LIN {X 0,Y 566.661,Z 389.019,A -85,B 0,C 180,E1 -2630.32,E2 -2630.32} C_VEL
LIN {X 0,Y 566.806,Z 374.387,A -85,B 0,C 180,E1 -2632.99,E2 -2632.99} C_VEL
LIN {X 0,Y 566.858,Z 367.103,A -85,B 0,C 180,E1 -2634.345,E2 -2634.345} C_VEL
LIN {X 0,Y 566.237,Z 363.511,A -85,B 0,C 180,E1 -2635.093,E2 -2635.093} C_VEL
LIN {X 0,Y 566.232,Z 363.455,A -85,B 0,C 180,E1 -2638.141,E2 -2638.141} C_VEL
LIN {X 0,Y 566.19,Z 363.456,A -85,B 0,C 180,E1 -2640.592,E2 -2640.592} C_VEL
LIN {X 0,Y 566.231,Z 363.447,A -85,B 0,C 180,E1 -2643.101,E2 -2643.101} C_VEL
LIN {X 0,Y 566.215,Z 363.454,A -85,B 0,C 180,E1 -2645.688,E2 -2645.688} C_VEL
LIN {X 0,Y 566.218,Z 363.451,A -85,B 0,C 180,E1 -2648.558,E2 -2648.558} C_VEL
LIN {X 0,Y 566.213,Z 363.446,A -85,B 0,C 180,E1 -2651.136,E2 -2651.136} C_VEL
LIN {X 0,Y 566.198,Z 363.46,A -85,B 0,C 180,E1 -2654.035,E2 -2654.035} C_VEL
LIN {X 0,Y 566.206,Z 363.45,A -85,B 0,C 180,E1 -2657.082,E2 -2657.082} C_VEL
LIN {X 0,Y 566.228,Z 363.455,A -85,B 0,C 180,E1 -2659.802,E2 -2659.802} C_VEL
LIN {X 0,Y 566.199,Z 363.452,A -85,B 0,C 180,E1 -2662.599,E2 -2662.599} C_VEL
LIN {X 0,Y 566.209,Z 363.449,A -85,B 0,C 180,E1 -2665.182,E2 -2665.182} C_VEL
LIN {X 0,Y 566.235,Z 363.453,A -85,B 0,C 180,E1 -2667.743,E2 -2667.743} C_VEL
LIN {X 0,Y 566.228,Z 363.45,A -85,B 0,C 180,E1 -2670.323,E2 -2670.323} C_VEL
LIN {X 0,Y 566.218,Z 363.446,A -85,B 0,C 180,E1 -2672.661,E2 -2672.661} C_VEL
LIN {X 0,Y 566.235,Z 363.445,A -85,B 0,C 180,E1 -2675.039,E2 -2675.039} C_VEL
LIN {X 0,Y 566.194,Z 363.455,A -85,B 0,C 180,E1 -2678.137,E2 -2678.137} C_VEL
LIN {X 0,Y 566.235,Z 363.443,A -85,B 0,C 180,E1 -2680.611,E2 -2680.611} C_VEL
LIN {X 0,Y 566.219,Z 363.45,A -85,B 0,C 180,E1 -2683.412,E2 -2683.412} C_VEL
LIN {X 0,Y 566.197,Z 363.452,A -85,B 0,C 180,E1 -2686.358,E2 -2686.358} C_VEL
LIN {X 0,Y 566.232,Z 363.445,A -85,B 0,C 180,E1 -2688.675,E2 -2688.675} C_VEL
LIN {X 0,Y 566.232,Z 363.446,A -85,B 0,C 180,E1 -2691.434,E2 -2691.434} C_VEL
LIN {X 0,Y 566.258,Z 363.445,A -85,B 0,C 180,E1 -2694.301,E2 -2694.301} C_VEL
LIN {X 0,Y 566.278,Z 363.445,A -85,B 0,C 180,E1 -2697.866,E2 -2697.866} C_VEL
LIN {X 0,Y 566.302,Z 363.433,A -85,B 0,C 180,E1 -2700.711,E2 -2700.711} C_VEL
LIN {X 0,Y 566.273,Z 363.441,A -85,B 0,C 180,E1 -2702.845,E2 -2702.845} C_VEL
LIN {X 0,Y 566.256,Z 363.452,A -85,B 0,C 180,E1 -2705.698,E2 -2705.698} C_VEL
LIN {X 0,Y 566.23,Z 363.444,A -85,B 0,C 180,E1 -2708.565,E2 -2708.565} C_VEL
LIN {X 0,Y 566.238,Z 363.45,A -85,B 0,C 180,E1 -2711.454,E2 -2711.454} C_VEL
LIN {X 0,Y 566.231,Z 363.447,A -85,B 0,C 180,E1 -2714.506,E2 -2714.506} C_VEL
LIN {X 0,Y 566.197,Z 363.457,A -85,B 0,C 180,E1 -2717.331,E2 -2717.331} C_VEL
LIN {X 0,Y 566.211,Z 363.447,A -85,B 0,C 180,E1 -2720.337,E2 -2720.337} C_VEL
LIN {X 0,Y 566.185,Z 363.462,A -85,B 0,C 180,E1 -2723.404,E2 -2723.404} C_VEL
LIN {X 0,Y 566.221,Z 363.451,A -85,B 0,C 180,E1 -2725.748,E2 -2725.748} C_VEL
LIN {X 0,Y 566.213,Z 363.453,A -85,B 0,C 180,E1 -2727.49,E2 -2727.49} C_VEL
LIN {X 0,Y 565.533,Z 363.534,A -85,B 0,C 180,E1 -2728.084,E2 -2728.084} C_VEL
LIN {X 0,Y 562.662,Z 363.893,A -85,B 0,C 180,E1 -2729.047,E2 -2729.047} C_VEL
LIN {X 0,Y 560.248,Z 364.196,A -85,B 0,C 180,E1 -2729.823,E2 -2729.823} C_VEL
LIN {X 0,Y 559.221,Z 364.321,A -85,B 0,C 180,E1 -2730.421,E2 -2730.421} C_VEL
LIN {X 0,Y 559.142,Z 364.331,A -85,B 0,C 180,E1 -2730.624,E2 -2730.624} C_VEL
LIN {X 0,Y 559.161,Z 364.332,A -85,B 0,C 180,E1 -2733.574,E2 -2733.574} C_VEL
LIN {X 0,Y 559.165,Z 364.327,A -85,B 0,C 180,E1 -2736.448,E2 -2736.448} C_VEL
LIN {X 0,Y 559.174,Z 364.33,A -85,B 0,C 180,E1 -2738.934,E2 -2738.934} C_VEL
LIN {X 0,Y 559.188,Z 364.328,A -85,B 0,C 180,E1 -2741.767,E2 -2741.767} C_VEL
LIN {X 0,Y 559.136,Z 364.333,A -85,B 0,C 180,E1 -2744.739,E2 -2744.739} C_VEL
LIN {X 0,Y 559.169,Z 364.321,A -85,B 0,C 180,E1 -2747.863,E2 -2747.863} C_VEL
LIN {X 0,Y 559.182,Z 364.324,A -85,B 0,C 180,E1 -2750.135,E2 -2750.135} C_VEL
LIN {X 0,Y 559.144,Z 364.335,A -85,B 0,C 180,E1 -2752.892,E2 -2752.892} C_VEL
LIN {X 0,Y 559.154,Z 364.331,A -85,B 0,C 180,E1 -2755.556,E2 -2755.556} C_VEL
LIN {X 0,Y 559.168,Z 364.328,A -85,B 0,C 180,E1 -2758.138,E2 -2758.138} C_VEL
LIN {X 0,Y 559.155,Z 364.328,A -85,B 0,C 180,E1 -2760.647,E2 -2760.647} C_VEL
LIN {X 0,Y 559.168,Z 364.337,A -85,B 0,C 180,E1 -2763.172,E2 -2763.172} C_VEL
LIN {X 0,Y 559.154,Z 364.335,A -85,B 0,C 180,E1 -2765.495,E2 -2765.495} C_VEL
LIN {X 0,Y 559.168,Z 364.33,A -85,B 0,C 180,E1 -2768.624,E2 -2768.624} C_VEL
LIN {X 0,Y 559.168,Z 364.335,A -85,B 0,C 180,E1 -2770.926,E2 -2770.926} C_VEL
LIN {X 0,Y 559.164,Z 364.329,A -85,B 0,C 180,E1 -2773.948,E2 -2773.948} C_VEL
LIN {X 0,Y 559.17,Z 364.328,A -85,B 0,C 180,E1 -2776.184,E2 -2776.184} C_VEL
LIN {X 0,Y 559.193,Z 364.334,A -85,B 0,C 180,E1 -2779.133,E2 -2779.133} C_VEL
LIN {X 0,Y 559.201,Z 364.324,A -85,B 0,C 180,E1 -2782.053,E2 -2782.053} C_VEL
LIN {X 0,Y 559.252,Z 364.326,A -85,B 0,C 180,E1 -2784.953,E2 -2784.953} C_VEL
LIN {X 0,Y 559.253,Z 364.318,A -85,B 0,C 180,E1 -2787.839,E2 -2787.839} C_VEL
LIN {X 0,Y 559.27,Z 364.321,A -85,B 0,C 180,E1 -2790.72,E2 -2790.72} C_VEL
LIN {X 0,Y 559.235,Z 364.328,A -85,B 0,C 180,E1 -2792.881,E2 -2792.881} C_VEL
LIN {X 0,Y 559.235,Z 364.32,A -85,B 0,C 180,E1 -2795.77,E2 -2795.77} C_VEL
LIN {X 0,Y 559.188,Z 364.332,A -85,B 0,C 180,E1 -2798.674,E2 -2798.674} C_VEL
LIN {X 0,Y 559.202,Z 364.325,A -85,B 0,C 180,E1 -2801.6,E2 -2801.6} C_VEL
LIN {X 0,Y 559.196,Z 364.33,A -85,B 0,C 180,E1 -2804.595,E2 -2804.595} C_VEL
LIN {X 0,Y 559.159,Z 364.33,A -85,B 0,C 180,E1 -2807.556,E2 -2807.556} C_VEL
LIN {X 0,Y 559.168,Z 364.328,A -85,B 0,C 180,E1 -2809.837,E2 -2809.837} C_VEL
LIN {X 0,Y 559.137,Z 364.333,A -85,B 0,C 180,E1 -2812.152,E2 -2812.152} C_VEL
LIN {X 0,Y 559.175,Z 364.331,A -85,B 0,C 180,E1 -2815.187,E2 -2815.187} C_VEL
LIN {X 0,Y 559.19,Z 364.325,A -85,B 0,C 180,E1 -2817.711,E2 -2817.711} C_VEL
LIN {X 0,Y 559.164,Z 364.327,A -85,B 0,C 180,E1 -2820.181,E2 -2820.181} C_VEL
LIN {X 0,Y 559.17,Z 364.336,A -85,B 0,C 180,E1 -2822.714,E2 -2822.714} C_VEL
LIN {X 0,Y 559.154,Z 364.328,A -85,B 0,C 180,E1 -2825.321,E2 -2825.321} C_VEL
LIN {X 0,Y 559.13,Z 364.333,A -85,B 0,C 180,E1 -2828.017,E2 -2828.017} C_VEL
LIN {X 0,Y 559.169,Z 364.328,A -85,B 0,C 180,E1 -2830.81,E2 -2830.81} C_VEL
LIN {X 0,Y 559.137,Z 364.327,A -85,B 0,C 180,E1 -2833.733,E2 -2833.733} C_VEL
LIN {X 0,Y 559.165,Z 364.335,A -85,B 0,C 180,E1 -2836.8,E2 -2836.8} C_VEL
LIN {X 0,Y 559.17,Z 364.327,A -85,B 0,C 180,E1 -2839.189,E2 -2839.189} C_VEL
LIN {X 0,Y 559.128,Z 364.334,A -85,B 0,C 180,E1 -2841.983,E2 -2841.983} C_VEL
LIN {X 0,Y 559.152,Z 364.333,A -85,B 0,C 180,E1 -2844.783,E2 -2844.783} C_VEL
LIN {X 0,Y 559.168,Z 364.327,A -85,B 0,C 180,E1 -2847.361,E2 -2847.361} C_VEL
LIN {X 0,Y 559.182,Z 364.329,A -85,B 0,C 180,E1 -2850.135,E2 -2850.135} C_VEL
LIN {X 0,Y 559.175,Z 364.325,A -85,B 0,C 180,E1 -2853.17,E2 -2853.17} C_VEL
LIN {X 0,Y 559.15,Z 364.329,A -85,B 0,C 180,E1 -2855.495,E2 -2855.495} C_VEL
LIN {X 0,Y 559.171,Z 364.332,A -85,B 0,C 180,E1 -2858.624,E2 -2858.624} C_VEL
LIN {X 0,Y 559.165,Z 364.326,A -85,B 0,C 180,E1 -2860.927,E2 -2860.927} C_VEL
LIN {X 0,Y 559.166,Z 364.329,A -85,B 0,C 180,E1 -2863.948,E2 -2863.948} C_VEL
LIN {X 0,Y 559.167,Z 364.333,A -85,B 0,C 180,E1 -2866.184,E2 -2866.184} C_VEL
LIN {X 0,Y 559.189,Z 364.32,A -85,B 0,C 180,E1 -2869.134,E2 -2869.134} C_VEL
LIN {X 0,Y 559.201,Z 364.324,A -85,B 0,C 180,E1 -2872.054,E2 -2872.054} C_VEL
LIN {X 0,Y 559.252,Z 364.318,A -85,B 0,C 180,E1 -2874.954,E2 -2874.954} C_VEL
LIN {X 0,Y 559.248,Z 364.317,A -85,B 0,C 180,E1 -2877.84,E2 -2877.84} C_VEL
LIN {X 0,Y 559.27,Z 364.316,A -85,B 0,C 180,E1 -2880.72,E2 -2880.72} C_VEL
LIN {X 0,Y 559.238,Z 364.32,A -85,B 0,C 180,E1 -2882.882,E2 -2882.882} C_VEL
LIN {X 0,Y 559.225,Z 364.322,A -85,B 0,C 180,E1 -2885.771,E2 -2885.771} C_VEL
LIN {X 0,Y 559.187,Z 364.322,A -85,B 0,C 180,E1 -2888.675,E2 -2888.675} C_VEL
LIN {X 0,Y 559.2,Z 364.321,A -85,B 0,C 180,E1 -2891.601,E2 -2891.601} C_VEL
LIN {X 0,Y 559.194,Z 364.327,A -85,B 0,C 180,E1 -2894.596,E2 -2894.596} C_VEL
LIN {X 0,Y 559.159,Z 364.326,A -85,B 0,C 180,E1 -2897.557,E2 -2897.557} C_VEL
LIN {X 0,Y 559.17,Z 364.326,A -85,B 0,C 180,E1 -2899.838,E2 -2899.838} C_VEL
LIN {X 0,Y 559.139,Z 364.339,A -85,B 0,C 180,E1 -2902.153,E2 -2902.153} C_VEL
LIN {X 0,Y 559.175,Z 364.324,A -85,B 0,C 180,E1 -2905.188,E2 -2905.188} C_VEL
LIN {X 0,Y 559.191,Z 364.323,A -85,B 0,C 180,E1 -2907.712,E2 -2907.712} C_VEL
LIN {X 0,Y 559.165,Z 364.337,A -85,B 0,C 180,E1 -2910.182,E2 -2910.182} C_VEL
LIN {X 0,Y 559.173,Z 364.326,A -85,B 0,C 180,E1 -2912.715,E2 -2912.715} C_VEL
LIN {X 0,Y 559.154,Z 364.328,A -85,B 0,C 180,E1 -2915.323,E2 -2915.323} C_VEL
LIN {X 0,Y 559.133,Z 364.341,A -85,B 0,C 180,E1 -2918.018,E2 -2918.018} C_VEL
LIN {X 0,Y 559.174,Z 364.326,A -85,B 0,C 180,E1 -2920.811,E2 -2920.811} C_VEL
LIN {X 0,Y 559.161,Z 364.333,A -85,B 0,C 180,E1 -2923.732,E2 -2923.732} C_VEL
LIN {X 0,Y 559.145,Z 364.33,A -85,B 0,C 180,E1 -2926.804,E2 -2926.804} C_VEL
LIN {X 0,Y 559.176,Z 364.322,A -85,B 0,C 180,E1 -2929.19,E2 -2929.19} C_VEL
LIN {X 0,Y 559.135,Z 364.341,A -85,B 0,C 180,E1 -2931.983,E2 -2931.983} C_VEL
LIN {X 0,Y 559.16,Z 364.328,A -85,B 0,C 180,E1 -2934.784,E2 -2934.784} C_VEL
LIN {X 0,Y 559.174,Z 364.328,A -85,B 0,C 180,E1 -2937.362,E2 -2937.362} C_VEL
LIN {X 0,Y 559.19,Z 364.333,A -85,B 0,C 180,E1 -2940.136,E2 -2940.136} C_VEL
LIN {X 0,Y 559.173,Z 364.33,A -85,B 0,C 180,E1 -2943.173,E2 -2943.173} C_VEL
LIN {X 0,Y 559.217,Z 364.47,A -85,B 0,C 180,E1 -2944.806,E2 -2944.806} C_VEL
LIN {X 0,Y 559.95,Z 370.109,A -85,B 0,C 180,E1 -2945.927,E2 -2945.927} C_VEL
LIN {X 0,Y 559.706,Z 385.772,A -85,B 0,C 180,E1 -2948.839,E2 -2948.839} C_VEL
LIN {X 0,Y 559.513,Z 401.439,A -85,B 0,C 180,E1 -2951.699,E2 -2951.699} C_VEL
LIN {X 0,Y 559.289,Z 417.995,A -85,B 0,C 180,E1 -2954.7,E2 -2954.7} C_VEL
LIN {X 0,Y 559.265,Z 424.262,A -85,B 0,C 180,E1 -2955.793,E2 -2955.793} C_VEL
LIN {X 0,Y 559.601,Z 426.656,A -85,B 0,C 180,E1 -2955.87,E2 -2955.87} C_VEL
LIN {X 0,Y 560.307,Z 432.116,A -85,B 0,C 180,E1 -2955.959,E2 -2955.959} C_VEL
LIN {X 0,Y 560.066,Z 530.587,A -85,B 0,C 180,E1 -2957.246,E2 -2957.246} C_VEL
LIN {X 0,Y 559.99,Z 540.847,A -85,B 0,C 180,E1 -2957.474,E2 -2957.474} C_VEL
LIN {X 0,Y 559.833,Z 551.603,A -85,B 0,C 180,E1 -2957.816,E2 -2957.816} C_VEL
LIN {X 0,Y 559.708,Z 561.373,A -85,B 0,C 180,E1 -2958.227,E2 -2958.227} C_VEL
LIN {X 0,Y 559.611,Z 571.083,A -85,B 0,C 180,E1 -2958.74,E2 -2958.74} C_VEL
LIN {X 0,Y 559.427,Z 581.44,A -85,B 0,C 180,E1 -2959.413,E2 -2959.413} C_VEL
LIN {X 0,Y 559.288,Z 591.646,A -85,B 0,C 180,E1 -2960.233,E2 -2960.233} C_VEL
LIN {X 0,Y 559.132,Z 600.795,A -85,B 0,C 180,E1 -2961.143,E2 -2961.143} C_VEL
LIN {X 0,Y 559.052,Z 608.331,A -85,B 0,C 180,E1 -2962.052,E2 -2962.052} C_VEL
LIN {X 0,Y 558.937,Z 614.719,A -85,B 0,C 180,E1 -2962.977,E2 -2962.977} C_VEL
LIN {X 0,Y 558.908,Z 619.843,A -85,B 0,C 180,E1 -2963.865,E2 -2963.865} C_VEL
LIN {X 0,Y 558.798,Z 624.907,A -85,B 0,C 180,E1 -2964.949,E2 -2964.949} C_VEL
LIN {X 0,Y 558.843,Z 628.846,A -85,B 0,C 180,E1 -2966.034,E2 -2966.034} C_VEL
LIN {X 0,Y 558.799,Z 631.76,A -85,B 0,C 180,E1 -2967.117,E2 -2967.117} C_VEL
LIN {X 0,Y 558.745,Z 633.211,A -85,B 0,C 180,E1 -2967.838,E2 -2967.838} C_VEL
LIN {X 0,Y 558.741,Z 634.756,A -85,B 0,C 180,E1 -2969.28,E2 -2969.28} C_VEL
LIN {X 0,Y 558.74,Z 635,A -85,B 0,C 180,E1 -2970,E2 -2970} C_VEL
LIN {X 0,Y 558.745,Z 634.165,A -85,B 0,C 180,E1 -2971.442,E2 -2971.442} C_VEL
LIN {X 0,Y 558.745,Z 633.211,A -85,B 0,C 180,E1 -2972.163,E2 -2972.163} C_VEL
LIN {X 0,Y 558.836,Z 629.925,A -85,B 0,C 180,E1 -2973.605,E2 -2973.605} C_VEL
LIN {X 0,Y 558.826,Z 626.324,A -85,B 0,C 180,E1 -2974.689,E2 -2974.689} C_VEL
LIN {X 0,Y 558.929,Z 621.629,A -85,B 0,C 180,E1 -2975.773,E2 -2975.773} C_VEL
LIN {X 0,Y 558.931,Z 615.912,A -85,B 0,C 180,E1 -2976.824,E2 -2976.824} C_VEL
LIN {X 0,Y 559.008,Z 609.635,A -85,B 0,C 180,E1 -2977.768,E2 -2977.768} C_VEL
LIN {X 0,Y 559.105,Z 602.365,A -85,B 0,C 180,E1 -2978.676,E2 -2978.676} C_VEL
LIN {X 0,Y 559.274,Z 593.602,A -85,B 0,C 180,E1 -2979.585,E2 -2979.585} C_VEL
LIN {X 0,Y 559.418,Z 582.721,A -85,B 0,C 180,E1 -2980.496,E2 -2980.496} C_VEL
LIN {X 0,Y 559.568,Z 572.533,A -85,B 0,C 180,E1 -2981.177,E2 -2981.177} C_VEL
LIN {X 0,Y 559.728,Z 561.753,A -85,B 0,C 180,E1 -2981.755,E2 -2981.755} C_VEL
LIN {X 0,Y 559.834,Z 551.591,A -85,B 0,C 180,E1 -2982.184,E2 -2982.184} C_VEL
LIN {X 0,Y 559.99,Z 540.83,A -85,B 0,C 180,E1 -2982.526,E2 -2982.526} C_VEL
LIN {X 0,Y 560.067,Z 530.561,A -85,B 0,C 180,E1 -2982.755,E2 -2982.755} C_VEL
LIN {X 0,Y 560.217,Z 430.294,A -85,B 0,C 180,E1 -2984.067,E2 -2984.067} C_VEL
LIN {X 0,Y 559.279,Z 424.58,A -85,B 0,C 180,E1 -2984.184,E2 -2984.184} C_VEL
LIN {X 0,Y 559.23,Z 423.167,A -85,B 0,C 180,E1 -2984.371,E2 -2984.371} C_VEL
LIN {X 0,Y 559.436,Z 406.941,A -85,B 0,C 180,E1 -2987.299,E2 -2987.299} C_VEL
LIN {X 0,Y 559.659,Z 389.957,A -85,B 0,C 180,E1 -2990.394,E2 -2990.394} C_VEL
LIN {X 0,Y 559.828,Z 376.374,A -85,B 0,C 180,E1 -2992.903,E2 -2992.903} C_VEL
LIN {X 0,Y 559.85,Z 368.049,A -85,B 0,C 180,E1 -2994.473,E2 -2994.473} C_VEL
LIN {X 0,Y 559.198,Z 364.383,A -85,B 0,C 180,E1 -2995.251,E2 -2995.251} C_VEL
LIN {X 0,Y 559.173,Z 364.334,A -85,B 0,C 180,E1 -2998.381,E2 -2998.381} C_VEL
LIN {X 0,Y 559.162,Z 364.329,A -85,B 0,C 180,E1 -3001.019,E2 -3001.019} C_VEL
LIN {X 0,Y 559.171,Z 364.335,A -85,B 0,C 180,E1 -3003.949,E2 -3003.949} C_VEL
LIN {X 0,Y 559.172,Z 364.33,A -85,B 0,C 180,E1 -3006.448,E2 -3006.448} C_VEL
LIN {X 0,Y 559.18,Z 364.325,A -85,B 0,C 180,E1 -3008.933,E2 -3008.933} C_VEL
LIN {X 0,Y 559.193,Z 364.326,A -85,B 0,C 180,E1 -3011.767,E2 -3011.767} C_VEL
LIN {X 0,Y 559.141,Z 364.331,A -85,B 0,C 180,E1 -3014.739,E2 -3014.739} C_VEL
LIN {X 0,Y 559.165,Z 364.328,A -85,B 0,C 180,E1 -3017.257,E2 -3017.257} C_VEL
LIN {X 0,Y 559.186,Z 364.33,A -85,B 0,C 180,E1 -3020.135,E2 -3020.135} C_VEL
LIN {X 0,Y 559.145,Z 364.33,A -85,B 0,C 180,E1 -3022.892,E2 -3022.892} C_VEL
LIN {X 0,Y 559.166,Z 364.332,A -85,B 0,C 180,E1 -3026.05,E2 -3026.05} C_VEL
LIN {X 0,Y 559.166,Z 364.327,A -85,B 0,C 180,E1 -3028.981,E2 -3028.981} C_VEL
LIN {X 0,Y 559.17,Z 364.332,A -85,B 0,C 180,E1 -3031.618,E2 -3031.618} C_VEL
LIN {X 0,Y 559.181,Z 364.331,A -85,B 0,C 180,E1 -3033.903,E2 -3033.903} C_VEL
LIN {X 0,Y 559.156,Z 364.329,A -85,B 0,C 180,E1 -3036.567,E2 -3036.567} C_VEL
LIN {X 0,Y 559.179,Z 364.328,A -85,B 0,C 180,E1 -3039.395,E2 -3039.395} C_VEL
LIN {X 0,Y 559.153,Z 364.332,A -85,B 0,C 180,E1 -3041.686,E2 -3041.686} C_VEL
LIN {X 0,Y 559.169,Z 364.333,A -85,B 0,C 180,E1 -3043.948,E2 -3043.948} C_VEL
LIN {X 0,Y 559.171,Z 364.329,A -85,B 0,C 180,E1 -3046.184,E2 -3046.184} C_VEL
LIN {X 0,Y 559.193,Z 364.323,A -85,B 0,C 180,E1 -3049.133,E2 -3049.133} C_VEL
LIN {X 0,Y 559.204,Z 364.325,A -85,B 0,C 180,E1 -3052.053,E2 -3052.053} C_VEL
LIN {X 0,Y 559.253,Z 364.317,A -85,B 0,C 180,E1 -3054.953,E2 -3054.953} C_VEL
LIN {X 0,Y 559.249,Z 364.321,A -85,B 0,C 180,E1 -3057.839,E2 -3057.839} C_VEL
LIN {X 0,Y 559.272,Z 364.308,A -85,B 0,C 180,E1 -3060.72,E2 -3060.72} C_VEL
LIN {X 0,Y 559.24,Z 364.317,A -85,B 0,C 180,E1 -3062.881,E2 -3062.881} C_VEL
LIN {X 0,Y 559.226,Z 364.327,A -85,B 0,C 180,E1 -3065.77,E2 -3065.77} C_VEL
LIN {X 0,Y 559.189,Z 364.321,A -85,B 0,C 180,E1 -3068.674,E2 -3068.674} C_VEL
LIN {X 0,Y 559.202,Z 364.329,A -85,B 0,C 180,E1 -3071.6,E2 -3071.6} C_VEL
LIN {X 0,Y 559.196,Z 364.324,A -85,B 0,C 180,E1 -3074.595,E2 -3074.595} C_VEL
LIN {X 0,Y 559.157,Z 364.334,A -85,B 0,C 180,E1 -3077.557,E2 -3077.557} C_VEL
LIN {X 0,Y 559.169,Z 364.329,A -85,B 0,C 180,E1 -3079.837,E2 -3079.837} C_VEL
LIN {X 0,Y 559.138,Z 364.332,A -85,B 0,C 180,E1 -3082.152,E2 -3082.152} C_VEL
LIN {X 0,Y 559.176,Z 364.331,A -85,B 0,C 180,E1 -3085.187,E2 -3085.187} C_VEL
LIN {X 0,Y 559.191,Z 364.327,A -85,B 0,C 180,E1 -3087.711,E2 -3087.711} C_VEL
LIN {X 0,Y 559.142,Z 364.331,A -85,B 0,C 180,E1 -3090.624,E2 -3090.624} C_VEL
LIN {X 0,Y 558.483,Z 364.421,A -85,B 0,C 180,E1 -3091.226,E2 -3091.226} C_VEL
LIN {X 0,Y 555.621,Z 364.773,A -85,B 0,C 180,E1 -3092.202,E2 -3092.202} C_VEL
LIN {X 0,Y 553.207,Z 365.073,A -85,B 0,C 180,E1 -3092.987,E2 -3092.987} C_VEL
LIN {X 0,Y 552.186,Z 365.2,A -85,B 0,C 180,E1 -3093.594,E2 -3093.594} C_VEL
LIN {X 0,Y 552.111,Z 365.204,A -85,B 0,C 180,E1 -3093.8,E2 -3093.8} C_VEL
LIN {X 0,Y 552.108,Z 365.207,A -85,B 0,C 180,E1 -3096.746,E2 -3096.746} C_VEL
LIN {X 0,Y 552.13,Z 365.209,A -85,B 0,C 180,E1 -3099.527,E2 -3099.527} C_VEL
LIN {X 0,Y 552.127,Z 365.204,A -85,B 0,C 180,E1 -3102.425,E2 -3102.425} C_VEL
LIN {X 0,Y 552.093,Z 365.21,A -85,B 0,C 180,E1 -3105.563,E2 -3105.563} C_VEL
LIN {X 0,Y 552.134,Z 365.196,A -85,B 0,C 180,E1 -3108.676,E2 -3108.676} C_VEL
LIN {X 0,Y 552.116,Z 365.214,A -85,B 0,C 180,E1 -3111.411,E2 -3111.411} C_VEL
LIN {X 0,Y 552.11,Z 365.204,A -85,B 0,C 180,E1 -3114.158,E2 -3114.158} C_VEL
LIN {X 0,Y 552.119,Z 365.206,A -85,B 0,C 180,E1 -3116.815,E2 -3116.815} C_VEL
LIN {X 0,Y 552.111,Z 365.211,A -85,B 0,C 180,E1 -3119.391,E2 -3119.391} C_VEL
LIN {X 0,Y 552.122,Z 365.206,A -85,B 0,C 180,E1 -3121.903,E2 -3121.903} C_VEL
LIN {X 0,Y 552.152,Z 365.204,A -85,B 0,C 180,E1 -3124.649,E2 -3124.649} C_VEL
LIN {X 0,Y 552.093,Z 365.213,A -85,B 0,C 180,E1 -3127.549,E2 -3127.549} C_VEL
LIN {X 0,Y 552.154,Z 365.205,A -85,B 0,C 180,E1 -3130.674,E2 -3130.674} C_VEL
LIN {X 0,Y 552.114,Z 365.208,A -85,B 0,C 180,E1 -3133.737,E2 -3133.737} C_VEL
LIN {X 0,Y 552.133,Z 365.205,A -85,B 0,C 180,E1 -3136.004,E2 -3136.004} C_VEL
LIN {X 0,Y 552.16,Z 365.209,A -85,B 0,C 180,E1 -3138.993,E2 -3138.993} C_VEL
LIN {X 0,Y 552.155,Z 365.202,A -85,B 0,C 180,E1 -3141.951,E2 -3141.951} C_VEL
LIN {X 0,Y 552.228,Z 365.201,A -85,B 0,C 180,E1 -3144.889,E2 -3144.889} C_VEL
LIN {X 0,Y 552.224,Z 365.194,A -85,B 0,C 180,E1 -3147.812,E2 -3147.812} C_VEL
LIN {X 0,Y 552.24,Z 365.197,A -85,B 0,C 180,E1 -3150.729,E2 -3150.729} C_VEL
LIN {X 0,Y 552.202,Z 365.204,A -85,B 0,C 180,E1 -3152.918,E2 -3152.918} C_VEL
LIN {X 0,Y 552.206,Z 365.196,A -85,B 0,C 180,E1 -3155.844,E2 -3155.844} C_VEL
LIN {X 0,Y 552.159,Z 365.209,A -85,B 0,C 180,E1 -3158.785,E2 -3158.785} C_VEL
LIN {X 0,Y 552.159,Z 365.202,A -85,B 0,C 180,E1 -3161.75,E2 -3161.75} C_VEL
LIN {X 0,Y 552.133,Z 365.212,A -85,B 0,C 180,E1 -3164.748,E2 -3164.748} C_VEL
LIN {X 0,Y 552.111,Z 365.208,A -85,B 0,C 180,E1 -3167.788,E2 -3167.788} C_VEL
LIN {X 0,Y 552.127,Z 365.206,A -85,B 0,C 180,E1 -3170.101,E2 -3170.101} C_VEL
LIN {X 0,Y 552.091,Z 365.214,A -85,B 0,C 180,E1 -3172.45,E2 -3172.45} C_VEL
LIN {X 0,Y 552.152,Z 365.204,A -85,B 0,C 180,E1 -3175.351,E2 -3175.351} C_VEL
LIN {X 0,Y 552.122,Z 365.206,A -85,B 0,C 180,E1 -3178.097,E2 -3178.097} C_VEL
LIN {X 0,Y 552.109,Z 365.211,A -85,B 0,C 180,E1 -3180.608,E2 -3180.608} C_VEL
LIN {X 0,Y 552.117,Z 365.206,A -85,B 0,C 180,E1 -3183.185,E2 -3183.185} C_VEL
LIN {X 0,Y 552.108,Z 365.204,A -85,B 0,C 180,E1 -3185.841,E2 -3185.841} C_VEL
LIN {X 0,Y 552.12,Z 365.208,A -85,B 0,C 180,E1 -3189.062,E2 -3189.062} C_VEL
LIN {X 0,Y 552.131,Z 365.196,A -85,B 0,C 180,E1 -3191.444,E2 -3191.444} C_VEL
LIN {X 0,Y 552.089,Z 365.212,A -85,B 0,C 180,E1 -3194.532,E2 -3194.532} C_VEL
LIN {X 0,Y 552.124,Z 365.204,A -85,B 0,C 180,E1 -3197.584,E2 -3197.584} C_VEL
LIN {X 0,Y 552.127,Z 365.209,A -85,B 0,C 180,E1 -3200.473,E2 -3200.473} C_VEL
LIN {X 0,Y 552.107,Z 365.207,A -85,B 0,C 180,E1 -3203.316,E2 -3203.316} C_VEL
LIN {X 0,Y 552.132,Z 365.201,A -85,B 0,C 180,E1 -3205.94,E2 -3205.94} C_VEL
LIN {X 0,Y 552.111,Z 365.215,A -85,B 0,C 180,E1 -3208.541,E2 -3208.541} C_VEL
LIN {X 0,Y 552.119,Z 365.203,A -85,B 0,C 180,E1 -3211.437,E2 -3211.437} C_VEL
LIN {X 0,Y 552.13,Z 365.208,A -85,B 0,C 180,E1 -3214.356,E2 -3214.356} C_VEL
LIN {X 0,Y 552.103,Z 365.213,A -85,B 0,C 180,E1 -3216.759,E2 -3216.759} C_VEL
LIN {X 0,Y 552.12,Z 365.203,A -85,B 0,C 180,E1 -3219.12,E2 -3219.12} C_VEL
LIN {X 0,Y 552.125,Z 365.2,A -85,B 0,C 180,E1 -3221.445,E2 -3221.445} C_VEL
LIN {X 0,Y 552.115,Z 365.205,A -85,B 0,C 180,E1 -3223.738,E2 -3223.738} C_VEL
LIN {X 0,Y 552.13,Z 365.207,A -85,B 0,C 180,E1 -3226.005,E2 -3226.005} C_VEL
LIN {X 0,Y 552.156,Z 365.197,A -85,B 0,C 180,E1 -3228.994,E2 -3228.994} C_VEL
LIN {X 0,Y 552.155,Z 365.2,A -85,B 0,C 180,E1 -3231.952,E2 -3231.952} C_VEL
LIN {X 0,Y 552.226,Z 365.194,A -85,B 0,C 180,E1 -3234.889,E2 -3234.889} C_VEL
LIN {X 0,Y 552.219,Z 365.192,A -85,B 0,C 180,E1 -3237.812,E2 -3237.812} C_VEL
LIN {X 0,Y 552.239,Z 365.191,A -85,B 0,C 180,E1 -3240.73,E2 -3240.73} C_VEL
LIN {X 0,Y 552.204,Z 365.196,A -85,B 0,C 180,E1 -3242.919,E2 -3242.919} C_VEL
LIN {X 0,Y 552.196,Z 365.198,A -85,B 0,C 180,E1 -3245.844,E2 -3245.844} C_VEL
LIN {X 0,Y 552.158,Z 365.196,A -85,B 0,C 180,E1 -3248.786,E2 -3248.786} C_VEL
LIN {X 0,Y 552.157,Z 365.2,A -85,B 0,C 180,E1 -3251.751,E2 -3251.751} C_VEL
LIN {X 0,Y 552.131,Z 365.205,A -85,B 0,C 180,E1 -3254.749,E2 -3254.749} C_VEL
LIN {X 0,Y 552.111,Z 365.206,A -85,B 0,C 180,E1 -3257.789,E2 -3257.789} C_VEL
LIN {X 0,Y 552.13,Z 365.207,A -85,B 0,C 180,E1 -3260.102,E2 -3260.102} C_VEL
LIN {X 0,Y 552.093,Z 365.214,A -85,B 0,C 180,E1 -3262.451,E2 -3262.451} C_VEL
LIN {X 0,Y 552.153,Z 365.199,A -85,B 0,C 180,E1 -3265.352,E2 -3265.352} C_VEL
LIN {X 0,Y 552.123,Z 365.209,A -85,B 0,C 180,E1 -3268.098,E2 -3268.098} C_VEL
LIN {X 0,Y 552.111,Z 365.209,A -85,B 0,C 180,E1 -3270.609,E2 -3270.609} C_VEL
LIN {X 0,Y 552.126,Z 365.202,A -85,B 0,C 180,E1 -3273.186,E2 -3273.186} C_VEL
LIN {X 0,Y 552.11,Z 365.21,A -85,B 0,C 180,E1 -3275.842,E2 -3275.842} C_VEL
LIN {X 0,Y 552.123,Z 365.203,A -85,B 0,C 180,E1 -3279.063,E2 -3279.063} C_VEL
LIN {X 0,Y 552.138,Z 365.204,A -85,B 0,C 180,E1 -3281.445,E2 -3281.445} C_VEL
LIN {X 0,Y 552.095,Z 365.21,A -85,B 0,C 180,E1 -3284.533,E2 -3284.533} C_VEL
LIN {X 0,Y 552.13,Z 365.207,A -85,B 0,C 180,E1 -3287.585,E2 -3287.585} C_VEL
LIN {X 0,Y 552.134,Z 365.206,A -85,B 0,C 180,E1 -3290.474,E2 -3290.474} C_VEL
LIN {X 0,Y 552.115,Z 365.207,A -85,B 0,C 180,E1 -3293.316,E2 -3293.316} C_VEL
LIN {X 0,Y 552.132,Z 365.213,A -85,B 0,C 180,E1 -3295.94,E2 -3295.94} C_VEL
LIN {X 0,Y 552.12,Z 365.208,A -85,B 0,C 180,E1 -3298.541,E2 -3298.541} C_VEL
LIN {X 0,Y 552.128,Z 365.209,A -85,B 0,C 180,E1 -3301.438,E2 -3301.438} C_VEL
LIN {X 0,Y 552.182,Z 365.271,A -85,B 0,C 180,E1 -3304.595,E2 -3304.595} C_VEL
LIN {X 0,Y 553.014,Z 371.056,A -85,B 0,C 180,E1 -3305.805,E2 -3305.805} C_VEL
LIN {X 0,Y 552.721,Z 386.682,A -85,B 0,C 180,E1 -3308.754,E2 -3308.754} C_VEL
LIN {X 0,Y 552.52,Z 403.419,A -85,B 0,C 180,E1 -3311.843,E2 -3311.843} C_VEL
LIN {X 0,Y 552.261,Z 421.1,A -85,B 0,C 180,E1 -3315.067,E2 -3315.067} C_VEL
LIN {X 0,Y 552.24,Z 424.435,A -85,B 0,C 180,E1 -3315.621,E2 -3315.621} C_VEL
LIN {X 0,Y 553.32,Z 430.71,A -85,B 0,C 180,E1 -3315.759,E2 -3315.759} C_VEL
LIN {X 0,Y 553.154,Z 530.532,A -85,B 0,C 180,E1 -3317.084,E2 -3317.084} C_VEL
LIN {X 0,Y 553.073,Z 540.812,A -85,B 0,C 180,E1 -3317.315,E2 -3317.315} C_VEL
LIN {X 0,Y 552.931,Z 550.567,A -85,B 0,C 180,E1 -3317.624,E2 -3317.624} C_VEL
LIN {X 0,Y 552.779,Z 560.151,A -85,B 0,C 180,E1 -3318.02,E2 -3318.02} C_VEL
LIN {X 0,Y 552.666,Z 569.69,A -85,B 0,C 180,E1 -3318.516,E2 -3318.516} C_VEL
LIN {X 0,Y 552.483,Z 578.805,A -85,B 0,C 180,E1 -3319.093,E2 -3319.093} C_VEL
LIN {X 0,Y 552.337,Z 587.293,A -85,B 0,C 180,E1 -3319.739,E2 -3319.739} C_VEL
LIN {X 0,Y 552.22,Z 595.44,A -85,B 0,C 180,E1 -3320.477,E2 -3320.477} C_VEL
LIN {X 0,Y 552.07,Z 602.358,A -85,B 0,C 180,E1 -3321.213,E2 -3321.213} C_VEL
LIN {X 0,Y 551.959,Z 609.628,A -85,B 0,C 180,E1 -3322.133,E2 -3322.133} C_VEL
LIN {X 0,Y 551.86,Z 615.688,A -85,B 0,C 180,E1 -3323.051,E2 -3323.051} C_VEL
LIN {X 0,Y 551.835,Z 620.409,A -85,B 0,C 180,E1 -3323.902,E2 -3323.902} C_VEL
LIN {X 0,Y 551.723,Z 624.901,A -85,B 0,C 180,E1 -3324.885,E2 -3324.885} C_VEL
LIN {X 0,Y 551.763,Z 628.839,A -85,B 0,C 180,E1 -3325.983,E2 -3325.983} C_VEL
LIN {X 0,Y 551.723,Z 631.752,A -85,B 0,C 180,E1 -3327.08,E2 -3327.08} C_VEL
LIN {X 0,Y 551.656,Z 633.213,A -85,B 0,C 180,E1 -3327.81,E2 -3327.81} C_VEL
LIN {X 0,Y 551.641,Z 634.747,A -85,B 0,C 180,E1 -3329.27,E2 -3329.27} C_VEL
LIN {X 0,Y 551.64,Z 635,A -85,B 0,C 180,E1 -3330,E2 -3330} C_VEL
LIN {X 0,Y 551.645,Z 634.157,A -85,B 0,C 180,E1 -3331.46,E2 -3331.46} C_VEL
LIN {X 0,Y 551.656,Z 633.212,A -85,B 0,C 180,E1 -3332.191,E2 -3332.191} C_VEL
LIN {X 0,Y 551.75,Z 629.918,A -85,B 0,C 180,E1 -3333.652,E2 -3333.652} C_VEL
LIN {X 0,Y 551.725,Z 626.318,A -85,B 0,C 180,E1 -3334.75,E2 -3334.75} C_VEL
LIN {X 0,Y 551.86,Z 621.621,A -85,B 0,C 180,E1 -3335.848,E2 -3335.848} C_VEL
LIN {X 0,Y 551.864,Z 617.639,A -85,B 0,C 180,E1 -3336.619,E2 -3336.619} C_VEL
LIN {X 0,Y 551.949,Z 610.931,A -85,B 0,C 180,E1 -3337.683,E2 -3337.683} C_VEL
LIN {X 0,Y 552.068,Z 603.909,A -85,B 0,C 180,E1 -3338.603,E2 -3338.603} C_VEL
LIN {X 0,Y 552.162,Z 597.279,A -85,B 0,C 180,E1 -3339.34,E2 -3339.34} C_VEL
LIN {X 0,Y 552.297,Z 588.383,A -85,B 0,C 180,E1 -3340.17,E2 -3340.17} C_VEL
LIN {X 0,Y 552.475,Z 580.109,A -85,B 0,C 180,E1 -3340.815,E2 -3340.815} C_VEL
LIN {X 0,Y 552.634,Z 570.732,A -85,B 0,C 180,E1 -3341.424,E2 -3341.424} C_VEL
LIN {X 0,Y 552.781,Z 561.34,A -85,B 0,C 180,E1 -3341.923,E2 -3341.923} C_VEL
LIN {X 0,Y 552.883,Z 551.563,A -85,B 0,C 180,E1 -3342.34,E2 -3342.34} C_VEL
LIN {X 0,Y 553.074,Z 540.796,A -85,B 0,C 180,E1 -3342.685,E2 -3342.685} C_VEL
LIN {X 0,Y 553.143,Z 530.507,A -85,B 0,C 180,E1 -3342.917,E2 -3342.917} C_VEL
LIN {X 0,Y 553.414,Z 433.919,A -85,B 0,C 180,E1 -3344.196,E2 -3344.196} C_VEL
LIN {X 0,Y 552.94,Z 428.646,A -85,B 0,C 180,E1 -3344.278,E2 -3344.278} C_VEL
LIN {X 0,Y 552.241,Z 424.427,A -85,B 0,C 180,E1 -3344.379,E2 -3344.379} C_VEL
LIN {X 0,Y 552.274,Z 417.993,A -85,B 0,C 180,E1 -3345.5,E2 -3345.5} C_VEL
LIN {X 0,Y 552.5,Z 402.371,A -85,B 0,C 180,E1 -3348.35,E2 -3348.35} C_VEL
LIN {X 0,Y 552.741,Z 385.641,A -85,B 0,C 180,E1 -3351.441,E2 -3351.441} C_VEL
LIN {X 0,Y 552.979,Z 370.038,A -85,B 0,C 180,E1 -3354.397,E2 -3354.397} C_VEL
LIN {X 0,Y 552.174,Z 365.283,A -85,B 0,C 180,E1 -3355.38,E2 -3355.38} C_VEL
LIN {X 0,Y 552.129,Z 365.212,A -85,B 0,C 180,E1 -3358.097,E2 -3358.097} C_VEL
LIN {X 0,Y 552.112,Z 365.21,A -85,B 0,C 180,E1 -3360.608,E2 -3360.608} C_VEL
LIN {X 0,Y 552.125,Z 365.204,A -85,B 0,C 180,E1 -3363.185,E2 -3363.185} C_VEL
LIN {X 0,Y 552.116,Z 365.212,A -85,B 0,C 180,E1 -3365.841,E2 -3365.841} C_VEL
LIN {X 0,Y 552.128,Z 365.204,A -85,B 0,C 180,E1 -3369.061,E2 -3369.061} C_VEL
LIN {X 0,Y 552.141,Z 365.2,A -85,B 0,C 180,E1 -3371.444,E2 -3371.444} C_VEL
LIN {X 0,Y 552.096,Z 365.21,A -85,B 0,C 180,E1 -3374.531,E2 -3374.531} C_VEL
LIN {X 0,Y 552.132,Z 365.208,A -85,B 0,C 180,E1 -3377.584,E2 -3377.584} C_VEL
LIN {X 0,Y 552.135,Z 365.204,A -85,B 0,C 180,E1 -3380.473,E2 -3380.473} C_VEL
LIN {X 0,Y 552.112,Z 365.208,A -85,B 0,C 180,E1 -3383.316,E2 -3383.316} C_VEL
LIN {X 0,Y 552.128,Z 365.209,A -85,B 0,C 180,E1 -3385.939,E2 -3385.939} C_VEL
LIN {X 0,Y 552.119,Z 365.206,A -85,B 0,C 180,E1 -3388.54,E2 -3388.54} C_VEL
LIN {X 0,Y 552.126,Z 365.207,A -85,B 0,C 180,E1 -3391.437,E2 -3391.437} C_VEL
LIN {X 0,Y 552.13,Z 365.204,A -85,B 0,C 180,E1 -3394.355,E2 -3394.355} C_VEL
LIN {X 0,Y 552.109,Z 365.206,A -85,B 0,C 180,E1 -3396.758,E2 -3396.758} C_VEL
LIN {X 0,Y 552.12,Z 365.205,A -85,B 0,C 180,E1 -3399.119,E2 -3399.119} C_VEL
LIN {X 0,Y 552.129,Z 365.203,A -85,B 0,C 180,E1 -3401.444,E2 -3401.444} C_VEL
LIN {X 0,Y 552.119,Z 365.211,A -85,B 0,C 180,E1 -3403.737,E2 -3403.737} C_VEL
LIN {X 0,Y 552.135,Z 365.208,A -85,B 0,C 180,E1 -3406.004,E2 -3406.004} C_VEL
LIN {X 0,Y 552.161,Z 365.198,A -85,B 0,C 180,E1 -3408.993,E2 -3408.993} C_VEL
LIN {X 0,Y 552.158,Z 365.204,A -85,B 0,C 180,E1 -3411.951,E2 -3411.951} C_VEL
LIN {X 0,Y 552.228,Z 365.192,A -85,B 0,C 180,E1 -3414.889,E2 -3414.889} C_VEL
LIN {X 0,Y 552.221,Z 365.197,A -85,B 0,C 180,E1 -3417.811,E2 -3417.811} C_VEL
LIN {X 0,Y 552.242,Z 365.183,A -85,B 0,C 180,E1 -3420.729,E2 -3420.729} C_VEL
LIN {X 0,Y 552.206,Z 365.193,A -85,B 0,C 180,E1 -3422.918,E2 -3422.918} C_VEL
LIN {X 0,Y 552.196,Z 365.201,A -85,B 0,C 180,E1 -3425.843,E2 -3425.843} C_VEL
LIN {X 0,Y 552.159,Z 365.197,A -85,B 0,C 180,E1 -3428.785,E2 -3428.785} C_VEL
LIN {X 0,Y 552.159,Z 365.205,A -85,B 0,C 180,E1 -3431.75,E2 -3431.75} C_VEL
LIN {X 0,Y 552.133,Z 365.204,A -85,B 0,C 180,E1 -3434.748,E2 -3434.748} C_VEL
LIN {X 0,Y 552.108,Z 365.207,A -85,B 0,C 180,E1 -3437.788,E2 -3437.788} C_VEL
LIN {X 0,Y 552.128,Z 365.203,A -85,B 0,C 180,E1 -3440.101,E2 -3440.101} C_VEL
LIN {X 0,Y 552.092,Z 365.208,A -85,B 0,C 180,E1 -3442.45,E2 -3442.45} C_VEL
LIN {X 0,Y 552.153,Z 365.209,A -85,B 0,C 180,E1 -3445.351,E2 -3445.351} C_VEL
LIN {X 0,Y 552.123,Z 365.203,A -85,B 0,C 180,E1 -3448.097,E2 -3448.097} C_VEL
LIN {X 0,Y 552.103,Z 365.208,A -85,B 0,C 180,E1 -3450.62,E2 -3450.62} C_VEL
LIN {X 0,Y 552.119,Z 365.211,A -85,B 0,C 180,E1 -3453.185,E2 -3453.185} C_VEL
LIN {X 0,Y 552.111,Z 365.204,A -85,B 0,C 180,E1 -3453.8,E2 -3453.8} C_VEL
LIN {X 0,Y 551.475,Z 365.284,A -85,B 0,C 180,E1 -3454.408,E2 -3454.408} C_VEL
LIN {X 0,Y 548.653,Z 365.643,A -85,B 0,C 180,E1 -3455.396,E2 -3455.396} C_VEL
LIN {X 0,Y 546.232,Z 365.941,A -85,B 0,C 180,E1 -3456.192,E2 -3456.192} C_VEL
LIN {X 0,Y 545.163,Z 366.073,A -85,B 0,C 180,E1 -3456.806,E2 -3456.806} C_VEL
LIN {X 0,Y 545.061,Z 366.088,A -85,B 0,C 180,E1 -3457.014,E2 -3457.014} C_VEL
LIN {X 0,Y 545.07,Z 366.081,A -85,B 0,C 180,E1 -3460.142,E2 -3460.142} C_VEL
LIN {X 0,Y 545.083,Z 366.087,A -85,B 0,C 180,E1 -3463.106,E2 -3463.106} C_VEL
LIN {X 0,Y 545.063,Z 366.08,A -85,B 0,C 180,E1 -3466.224,E2 -3466.224} C_VEL
LIN {X 0,Y 545.096,Z 366.074,A -85,B 0,C 180,E1 -3468.887,E2 -3468.887} C_VEL
LIN {X 0,Y 545.05,Z 366.089,A -85,B 0,C 180,E1 -3471.763,E2 -3471.763} C_VEL
LIN {X 0,Y 545.062,Z 366.082,A -85,B 0,C 180,E1 -3474.534,E2 -3474.534} C_VEL
LIN {X 0,Y 545.078,Z 366.089,A -85,B 0,C 180,E1 -3477.212,E2 -3477.212} C_VEL
LIN {X 0,Y 545.099,Z 366.078,A -85,B 0,C 180,E1 -3479.813,E2 -3479.813} C_VEL
LIN {X 0,Y 545.093,Z 366.085,A -85,B 0,C 180,E1 -3482.826,E2 -3482.826} C_VEL
LIN {X 0,Y 545.049,Z 366.09,A -85,B 0,C 180,E1 -3485.631,E2 -3485.631} C_VEL
LIN {X 0,Y 545.063,Z 366.09,A -85,B 0,C 180,E1 -3488.837,E2 -3488.837} C_VEL
LIN {X 0,Y 545.082,Z 366.091,A -85,B 0,C 180,E1 -3491.196,E2 -3491.196} C_VEL
LIN {X 0,Y 545.07,Z 366.088,A -85,B 0,C 180,E1 -3493.521,E2 -3493.521} C_VEL
LIN {X 0,Y 545.092,Z 366.083,A -85,B 0,C 180,E1 -3495.82,E2 -3495.82} C_VEL
LIN {X 0,Y 545.115,Z 366.085,A -85,B 0,C 180,E1 -3498.849,E2 -3498.849} C_VEL
LIN {X 0,Y 545.126,Z 366.079,A -85,B 0,C 180,E1 -3501.847,E2 -3501.847} C_VEL
LIN {X 0,Y 545.204,Z 366.075,A -85,B 0,C 180,E1 -3504.823,E2 -3504.823} C_VEL
LIN {X 0,Y 545.195,Z 366.07,A -85,B 0,C 180,E1 -3507.783,E2 -3507.783} C_VEL
LIN {X 0,Y 545.21,Z 366.073,A -85,B 0,C 180,E1 -3510.738,E2 -3510.738} C_VEL
LIN {X 0,Y 545.168,Z 366.08,A -85,B 0,C 180,E1 -3512.956,E2 -3512.956} C_VEL
LIN {X 0,Y 545.177,Z 366.072,A -85,B 0,C 180,E1 -3515.919,E2 -3515.919} C_VEL
LIN {X 0,Y 545.118,Z 366.087,A -85,B 0,C 180,E1 -3518.9,E2 -3518.9} C_VEL
LIN {X 0,Y 545.131,Z 366.077,A -85,B 0,C 180,E1 -3521.904,E2 -3521.904} C_VEL
LIN {X 0,Y 545.082,Z 366.091,A -85,B 0,C 180,E1 -3524.943,E2 -3524.943} C_VEL
LIN {X 0,Y 545.079,Z 366.084,A -85,B 0,C 180,E1 -3528.025,E2 -3528.025} C_VEL
LIN {X 0,Y 545.091,Z 366.085,A -85,B 0,C 180,E1 -3530.372,E2 -3530.372} C_VEL
LIN {X 0,Y 545.087,Z 366.083,A -85,B 0,C 180,E1 -3533.558,E2 -3533.558} C_VEL
LIN {X 0,Y 545.084,Z 366.083,A -85,B 0,C 180,E1 -3536,E2 -3536} C_VEL
LIN {X 0,Y 545.088,Z 366.086,A -85,B 0,C 180,E1 -3538.749,E2 -3538.749} C_VEL
LIN {X 0,Y 545.072,Z 366.084,A -85,B 0,C 180,E1 -3541.682,E2 -3541.682} C_VEL
LIN {X 0,Y 545.077,Z 366.084,A -85,B 0,C 180,E1 -3544.563,E2 -3544.563} C_VEL
LIN {X 0,Y 545.034,Z 366.09,A -85,B 0,C 180,E1 -3547.303,E2 -3547.303} C_VEL
LIN {X 0,Y 545.086,Z 366.082,A -85,B 0,C 180,E1 -3550.14,E2 -3550.14} C_VEL
LIN {X 0,Y 545.071,Z 366.082,A -85,B 0,C 180,E1 -3553.106,E2 -3553.106} C_VEL
LIN {X 0,Y 545.059,Z 366.088,A -85,B 0,C 180,E1 -3556.224,E2 -3556.224} C_VEL
LIN {X 0,Y 545.091,Z 366.084,A -85,B 0,C 180,E1 -3558.887,E2 -3558.887} C_VEL
LIN {X 0,Y 545.047,Z 366.087,A -85,B 0,C 180,E1 -3561.763,E2 -3561.763} C_VEL
LIN {X 0,Y 545.058,Z 366.091,A -85,B 0,C 180,E1 -3564.534,E2 -3564.534} C_VEL
LIN {X 0,Y 545.076,Z 366.084,A -85,B 0,C 180,E1 -3567.213,E2 -3567.213} C_VEL
LIN {X 0,Y 545.094,Z 366.081,A -85,B 0,C 180,E1 -3569.813,E2 -3569.813} C_VEL
LIN {X 0,Y 545.094,Z 366.082,A -85,B 0,C 180,E1 -3572.825,E2 -3572.825} C_VEL
LIN {X 0,Y 545.045,Z 366.086,A -85,B 0,C 180,E1 -3575.631,E2 -3575.631} C_VEL
LIN {X 0,Y 545.063,Z 366.085,A -85,B 0,C 180,E1 -3578.837,E2 -3578.837} C_VEL
LIN {X 0,Y 545.077,Z 366.078,A -85,B 0,C 180,E1 -3581.196,E2 -3581.196} C_VEL
LIN {X 0,Y 545.071,Z 366.082,A -85,B 0,C 180,E1 -3583.522,E2 -3583.522} C_VEL
LIN {X 0,Y 545.089,Z 366.082,A -85,B 0,C 180,E1 -3585.82,E2 -3585.82} C_VEL
LIN {X 0,Y 545.111,Z 366.075,A -85,B 0,C 180,E1 -3588.85,E2 -3588.85} C_VEL
LIN {X 0,Y 545.125,Z 366.074,A -85,B 0,C 180,E1 -3591.847,E2 -3591.847} C_VEL
LIN {X 0,Y 545.202,Z 366.07,A -85,B 0,C 180,E1 -3594.823,E2 -3594.823} C_VEL
LIN {X 0,Y 545.191,Z 366.067,A -85,B 0,C 180,E1 -3597.784,E2 -3597.784} C_VEL
LIN {X 0,Y 545.209,Z 366.066,A -85,B 0,C 180,E1 -3600.739,E2 -3600.739} C_VEL
LIN {X 0,Y 545.17,Z 366.072,A -85,B 0,C 180,E1 -3602.956,E2 -3602.956} C_VEL
LIN {X 0,Y 545.167,Z 366.075,A -85,B 0,C 180,E1 -3605.92,E2 -3605.92} C_VEL
LIN {X 0,Y 545.116,Z 366.071,A -85,B 0,C 180,E1 -3608.9,E2 -3608.9} C_VEL
LIN {X 0,Y 545.13,Z 366.077,A -85,B 0,C 180,E1 -3611.905,E2 -3611.905} C_VEL
LIN {X 0,Y 545.081,Z 366.082,A -85,B 0,C 180,E1 -3614.944,E2 -3614.944} C_VEL
LIN {X 0,Y 545.079,Z 366.084,A -85,B 0,C 180,E1 -3618.026,E2 -3618.026} C_VEL
LIN {X 0,Y 545.095,Z 366.086,A -85,B 0,C 180,E1 -3620.372,E2 -3620.372} C_VEL
LIN {X 0,Y 545.087,Z 366.082,A -85,B 0,C 180,E1 -3623.559,E2 -3623.559} C_VEL
LIN {X 0,Y 545.085,Z 366.086,A -85,B 0,C 180,E1 -3626.001,E2 -3626.001} C_VEL
LIN {X 0,Y 545.089,Z 366.082,A -85,B 0,C 180,E1 -3628.75,E2 -3628.75} C_VEL
LIN {X 0,Y 545.075,Z 366.086,A -85,B 0,C 180,E1 -3631.683,E2 -3631.683} C_VEL
LIN {X 0,Y 545.081,Z 366.083,A -85,B 0,C 180,E1 -3634.564,E2 -3634.564} C_VEL
LIN {X 0,Y 545.037,Z 366.088,A -85,B 0,C 180,E1 -3637.304,E2 -3637.304} C_VEL
LIN {X 0,Y 545.091,Z 366.088,A -85,B 0,C 180,E1 -3640.141,E2 -3640.141} C_VEL
LIN {X 0,Y 545.085,Z 366.081,A -85,B 0,C 180,E1 -3643.106,E2 -3643.106} C_VEL
LIN {X 0,Y 545.065,Z 366.09,A -85,B 0,C 180,E1 -3646.225,E2 -3646.225} C_VEL
LIN {X 0,Y 545.096,Z 366.075,A -85,B 0,C 180,E1 -3648.888,E2 -3648.888} C_VEL
LIN {X 0,Y 545.054,Z 366.091,A -85,B 0,C 180,E1 -3651.764,E2 -3651.764} C_VEL
LIN {X 0,Y 545.066,Z 366.086,A -85,B 0,C 180,E1 -3654.535,E2 -3654.535} C_VEL
LIN {X 0,Y 545.082,Z 366.082,A -85,B 0,C 180,E1 -3657.213,E2 -3657.213} C_VEL
LIN {X 0,Y 545.103,Z 366.087,A -85,B 0,C 180,E1 -3659.814,E2 -3659.814} C_VEL
LIN {X 0,Y 545.098,Z 366.084,A -85,B 0,C 180,E1 -3662.827,E2 -3662.827} C_VEL
LIN {X 0,Y 545.154,Z 366.198,A -85,B 0,C 180,E1 -3664.479,E2 -3664.479} C_VEL
LIN {X 0,Y 546.051,Z 372.003,A -85,B 0,C 180,E1 -3665.679,E2 -3665.679} C_VEL
LIN {X 0,Y 545.766,Z 386.546,A -85,B 0,C 180,E1 -3668.47,E2 -3668.47} C_VEL
LIN {X 0,Y 545.479,Z 401.192,A -85,B 0,C 180,E1 -3671.21,E2 -3671.21} C_VEL
LIN {X 0,Y 545.286,Z 415.817,A -85,B 0,C 180,E1 -3673.913,E2 -3673.913} C_VEL
LIN {X 0,Y 545.17,Z 424.194,A -85,B 0,C 180,E1 -3675.415,E2 -3675.415} C_VEL
LIN {X 0,Y 545.497,Z 426.377,A -85,B 0,C 180,E1 -3675.493,E2 -3675.493} C_VEL
LIN {X 0,Y 546.55,Z 433.728,A -85,B 0,C 180,E1 -3675.619,E2 -3675.619} C_VEL
LIN {X 0,Y 546.291,Z 529.156,A -85,B 0,C 180,E1 -3676.895,E2 -3676.895} C_VEL
LIN {X 0,Y 546.114,Z 539.057,A -85,B 0,C 180,E1 -3677.103,E2 -3677.103} C_VEL
LIN {X 0,Y 546.017,Z 549.03,A -85,B 0,C 180,E1 -3677.408,E2 -3677.408} C_VEL
LIN {X 0,Y 545.848,Z 559.368,A -85,B 0,C 180,E1 -3677.829,E2 -3677.829} C_VEL
LIN {X 0,Y 545.688,Z 568.612,A -85,B 0,C 180,E1 -3678.304,E2 -3678.304} C_VEL
LIN {X 0,Y 545.555,Z 577.481,A -85,B 0,C 180,E1 -3678.859,E2 -3678.859} C_VEL
LIN {X 0,Y 545.383,Z 586.184,A -85,B 0,C 180,E1 -3679.513,E2 -3679.513} C_VEL
LIN {X 0,Y 545.223,Z 593.583,A -85,B 0,C 180,E1 -3680.166,E2 -3680.166} C_VEL
LIN {X 0,Y 545.028,Z 602.347,A -85,B 0,C 180,E1 -3681.099,E2 -3681.099} C_VEL
LIN {X 0,Y 544.915,Z 609.618,A -85,B 0,C 180,E1 -3682.031,E2 -3682.031} C_VEL
LIN {X 0,Y 544.79,Z 615.679,A -85,B 0,C 180,E1 -3682.961,E2 -3682.961} C_VEL
LIN {X 0,Y 544.723,Z 619.644,A -85,B 0,C 180,E1 -3683.665,E2 -3683.665} C_VEL
LIN {X 0,Y 544.653,Z 624.895,A -85,B 0,C 180,E1 -3684.818,E2 -3684.818} C_VEL
LIN {X 0,Y 544.683,Z 628.832,A -85,B 0,C 180,E1 -3685.931,E2 -3685.931} C_VEL
LIN {X 0,Y 544.65,Z 631.744,A -85,B 0,C 180,E1 -3687.042,E2 -3687.042} C_VEL
LIN {X 0,Y 544.571,Z 633.214,A -85,B 0,C 180,E1 -3687.781,E2 -3687.781} C_VEL
LIN {X 0,Y 544.542,Z 634.74,A -85,B 0,C 180,E1 -3689.261,E2 -3689.261} C_VEL
LIN {X 0,Y 544.541,Z 635,A -85,B 0,C 180,E1 -3690,E2 -3690} C_VEL
LIN {X 0,Y 544.546,Z 634.15,A -85,B 0,C 180,E1 -3691.479,E2 -3691.479} C_VEL
LIN {X 0,Y 544.571,Z 633.213,A -85,B 0,C 180,E1 -3692.219,E2 -3692.219} C_VEL
LIN {X 0,Y 544.669,Z 629.911,A -85,B 0,C 180,E1 -3693.699,E2 -3693.699} C_VEL
LIN {X 0,Y 544.628,Z 626.311,A -85,B 0,C 180,E1 -3694.812,E2 -3694.812} C_VEL
LIN {X 0,Y 544.769,Z 621.613,A -85,B 0,C 180,E1 -3695.924,E2 -3695.924} C_VEL
LIN {X 0,Y 544.796,Z 616.763,A -85,B 0,C 180,E1 -3696.853,E2 -3696.853} C_VEL
LIN {X 0,Y 544.895,Z 610.92,A -85,B 0,C 180,E1 -3697.783,E2 -3697.783} C_VEL
LIN {X 0,Y 545.019,Z 603.898,A -85,B 0,C 180,E1 -3698.715,E2 -3698.715} C_VEL
LIN {X 0,Y 545.151,Z 597.267,A -85,B 0,C 180,E1 -3699.461,E2 -3699.461} C_VEL
LIN {X 0,Y 545.249,Z 589.465,A -85,B 0,C 180,E1 -3700.209,E2 -3700.209} C_VEL
LIN {X 0,Y 545.462,Z 581.404,A -85,B 0,C 180,E1 -3700.862,E2 -3700.862} C_VEL
LIN {X 0,Y 545.622,Z 573.284,A -85,B 0,C 180,E1 -3701.421,E2 -3701.421} C_VEL
LIN {X 0,Y 545.798,Z 563.29,A -85,B 0,C 180,E1 -3701.984,E2 -3701.984} C_VEL
LIN {X 0,Y 545.931,Z 552.801,A -85,B 0,C 180,E1 -3702.453,E2 -3702.453} C_VEL
LIN {X 0,Y 546.104,Z 542.482,A -85,B 0,C 180,E1 -3702.803,E2 -3702.803} C_VEL
LIN {X 0,Y 546.224,Z 531.773,A -85,B 0,C 180,E1 -3703.06,E2 -3703.06} C_VEL
LIN {X 0,Y 546.389,Z 507.207,A -85,B 0,C 180,E1 -3703.411,E2 -3703.411} C_VEL
LIN {X 0,Y 546.404,Z 431.433,A -85,B 0,C 180,E1 -3704.415,E2 -3704.415} C_VEL
LIN {X 0,Y 545.205,Z 424.421,A -85,B 0,C 180,E1 -3704.565,E2 -3704.565} C_VEL
LIN {X 0,Y 545.249,Z 418.946,A -85,B 0,C 180,E1 -3705.513,E2 -3705.513} C_VEL
LIN {X 0,Y 545.501,Z 403.281,A -85,B 0,C 180,E1 -3708.4,E2 -3708.4} C_VEL
LIN {X 0,Y 545.718,Z 387.624,A -85,B 0,C 180,E1 -3711.335,E2 -3711.335} C_VEL
LIN {X 0,Y 546.02,Z 373.925,A -85,B 0,C 180,E1 -3713.954,E2 -3713.954} C_VEL
LIN {X 0,Y 545.82,Z 369.94,A -85,B 0,C 180,E1 -3714.738,E2 -3714.738} C_VEL
LIN {X 0,Y 545.142,Z 366.161,A -85,B 0,C 180,E1 -3715.546,E2 -3715.546} C_VEL
LIN {X 0,Y 545.096,Z 366.084,A -85,B 0,C 180,E1 -3718.749,E2 -3718.749} C_VEL
LIN {X 0,Y 545.072,Z 366.085,A -85,B 0,C 180,E1 -3721.047,E2 -3721.047} C_VEL
LIN {X 0,Y 545.074,Z 366.086,A -85,B 0,C 180,E1 -3723.671,E2 -3723.671} C_VEL
LIN {X 0,Y 545.059,Z 366.089,A -85,B 0,C 180,E1 -3726.379,E2 -3726.379} C_VEL
LIN {X 0,Y 545.108,Z 366.08,A -85,B 0,C 180,E1 -3729.324,E2 -3729.324} C_VEL
LIN {X 0,Y 545.085,Z 366.089,A -85,B 0,C 180,E1 -3732.102,E2 -3732.102} C_VEL
LIN {X 0,Y 545.064,Z 366.084,A -85,B 0,C 180,E1 -3735.167,E2 -3735.167} C_VEL
LIN {X 0,Y 545.084,Z 366.091,A -85,B 0,C 180,E1 -3737.897,E2 -3737.897} C_VEL
LIN {X 0,Y 545.106,Z 366.078,A -85,B 0,C 180,E1 -3740.675,E2 -3740.675} C_VEL
LIN {X 0,Y 545.051,Z 366.091,A -85,B 0,C 180,E1 -3743.62,E2 -3743.62} C_VEL
LIN {X 0,Y 545.069,Z 366.084,A -85,B 0,C 180,E1 -3746.328,E2 -3746.328} C_VEL
LIN {X 0,Y 545.07,Z 366.083,A -85,B 0,C 180,E1 -3748.952,E2 -3748.952} C_VEL
LIN {X 0,Y 545.104,Z 366.083,A -85,B 0,C 180,E1 -3751.507,E2 -3751.507} C_VEL
LIN {X 0,Y 545.094,Z 366.079,A -85,B 0,C 180,E1 -3754.491,E2 -3754.491} C_VEL
LIN {X 0,Y 545.044,Z 366.088,A -85,B 0,C 180,E1 -3757.242,E2 -3757.242} C_VEL
LIN {X 0,Y 545.119,Z 366.073,A -85,B 0,C 180,E1 -3760.414,E2 -3760.414} C_VEL
LIN {X 0,Y 545.075,Z 366.084,A -85,B 0,C 180,E1 -3763.521,E2 -3763.521} C_VEL
LIN {X 0,Y 545.094,Z 366.088,A -85,B 0,C 180,E1 -3765.82,E2 -3765.82} C_VEL
LIN {X 0,Y 545.116,Z 366.074,A -85,B 0,C 180,E1 -3768.849,E2 -3768.849} C_VEL
LIN {X 0,Y 545.128,Z 366.081,A -85,B 0,C 180,E1 -3771.847,E2 -3771.847} C_VEL
LIN {X 0,Y 545.203,Z 366.067,A -85,B 0,C 180,E1 -3774.823,E2 -3774.823} C_VEL
LIN {X 0,Y 545.193,Z 366.072,A -85,B 0,C 180,E1 -3777.783,E2 -3777.783} C_VEL
LIN {X 0,Y 545.212,Z 366.058,A -85,B 0,C 180,E1 -3780.738,E2 -3780.738} C_VEL
LIN {X 0,Y 545.172,Z 366.069,A -85,B 0,C 180,E1 -3782.955,E2 -3782.955} C_VEL
LIN {X 0,Y 545.168,Z 366.075,A -85,B 0,C 180,E1 -3785.919,E2 -3785.919} C_VEL
LIN {X 0,Y 545.118,Z 366.074,A -85,B 0,C 180,E1 -3788.9,E2 -3788.9} C_VEL
LIN {X 0,Y 545.132,Z 366.078,A -85,B 0,C 180,E1 -3791.904,E2 -3791.904} C_VEL
LIN {X 0,Y 545.083,Z 366.083,A -85,B 0,C 180,E1 -3794.943,E2 -3794.943} C_VEL
LIN {X 0,Y 545.076,Z 366.08,A -85,B 0,C 180,E1 -3798.025,E2 -3798.025} C_VEL
LIN {X 0,Y 545.092,Z 366.077,A -85,B 0,C 180,E1 -3800.372,E2 -3800.372} C_VEL
LIN {X 0,Y 545.088,Z 366.089,A -85,B 0,C 180,E1 -3803.558,E2 -3803.558} C_VEL
LIN {X 0,Y 545.085,Z 366.08,A -85,B 0,C 180,E1 -3806,E2 -3806} C_VEL
LIN {X 0,Y 545.086,Z 366.079,A -85,B 0,C 180,E1 -3808.748,E2 -3808.748} C_VEL
LIN {X 0,Y 545.074,Z 366.088,A -85,B 0,C 180,E1 -3811.682,E2 -3811.682} C_VEL
LIN {X 0,Y 545.077,Z 366.078,A -85,B 0,C 180,E1 -3814.563,E2 -3814.563} C_VEL
LIN {X 0,Y 545.061,Z 366.088,A -85,B 0,C 180,E1 -3817.014,E2 -3817.014} C_VEL
LIN {X 0,Y 544.354,Z 366.182,A -85,B 0,C 180,E1 -3817.63,E2 -3817.63} C_VEL
LIN {X 0,Y 541.49,Z 366.536,A -85,B 0,C 180,E1 -3818.631,E2 -3818.631} C_VEL
LIN {X 0,Y 539.103,Z 366.832,A -85,B 0,C 180,E1 -3819.437,E2 -3819.437} C_VEL
LIN {X 0,Y 538.093,Z 366.951,A -85,B 0,C 180,E1 -3820.059,E2 -3820.059} C_VEL
LIN {X 0,Y 538.018,Z 366.959,A -85,B 0,C 180,E1 -3820.269,E2 -3820.269} C_VEL
LIN {X 0,Y 538.029,Z 366.964,A -85,B 0,C 180,E1 -3822.988,E2 -3822.988} C_VEL
LIN {X 0,Y 538.025,Z 366.957,A -85,B 0,C 180,E1 -3825.925,E2 -3825.925} C_VEL
LIN {X 0,Y 538.074,Z 366.953,A -85,B 0,C 180,E1 -3829.249,E2 -3829.249} C_VEL
LIN {X 0,Y 537.99,Z 366.966,A -85,B 0,C 180,E1 -3832.122,E2 -3832.122} C_VEL
LIN {X 0,Y 538.017,Z 366.963,A -85,B 0,C 180,E1 -3834.917,E2 -3834.917} C_VEL
LIN {X 0,Y 538.028,Z 366.965,A -85,B 0,C 180,E1 -3837.618,E2 -3837.618} C_VEL
LIN {X 0,Y 538.04,Z 366.956,A -85,B 0,C 180,E1 -3840.24,E2 -3840.24} C_VEL
LIN {X 0,Y 538.063,Z 366.96,A -85,B 0,C 180,E1 -3842.796,E2 -3842.796} C_VEL
LIN {X 0,Y 538.046,Z 366.967,A -85,B 0,C 180,E1 -3845.293,E2 -3845.293} C_VEL
LIN {X 0,Y 538.012,Z 366.964,A -85,B 0,C 180,E1 -3848.042,E2 -3848.042} C_VEL
LIN {X 0,Y 538.038,Z 366.967,A -85,B 0,C 180,E1 -3850.94,E2 -3850.94} C_VEL
LIN {X 0,Y 538.022,Z 366.97,A -85,B 0,C 180,E1 -3853.299,E2 -3853.299} C_VEL
LIN {X 0,Y 538.061,Z 366.96,A -85,B 0,C 180,E1 -3855.631,E2 -3855.631} C_VEL
LIN {X 0,Y 538.075,Z 366.961,A -85,B 0,C 180,E1 -3858.701,E2 -3858.701} C_VEL
LIN {X 0,Y 538.083,Z 366.957,A -85,B 0,C 180,E1 -3861.739,E2 -3861.739} C_VEL
LIN {X 0,Y 538.162,Z 366.951,A -85,B 0,C 180,E1 -3864.755,E2 -3864.755} C_VEL
LIN {X 0,Y 538.167,Z 366.946,A -85,B 0,C 180,E1 -3867.755,E2 -3867.755} C_VEL
LIN {X 0,Y 538.18,Z 366.949,A -85,B 0,C 180,E1 -3870.748,E2 -3870.748} C_VEL
LIN {X 0,Y 538.135,Z 366.957,A -85,B 0,C 180,E1 -3872.994,E2 -3872.994} C_VEL
LIN {X 0,Y 538.131,Z 366.95,A -85,B 0,C 180,E1 -3875.997,E2 -3875.997} C_VEL
LIN {X 0,Y 538.068,Z 366.965,A -85,B 0,C 180,E1 -3879.017,E2 -3879.017} C_VEL
LIN {X 0,Y 538.08,Z 366.956,A -85,B 0,C 180,E1 -3882.062,E2 -3882.062} C_VEL
LIN {X 0,Y 538.041,Z 366.966,A -85,B 0,C 180,E1 -3885.143,E2 -3885.143} C_VEL
LIN {X 0,Y 538.031,Z 366.963,A -85,B 0,C 180,E1 -3888.27,E2 -3888.27} C_VEL
LIN {X 0,Y 538.035,Z 366.968,A -85,B 0,C 180,E1 -3890.651,E2 -3890.651} C_VEL
LIN {X 0,Y 538.019,Z 366.963,A -85,B 0,C 180,E1 -3893.887,E2 -3893.887} C_VEL
LIN {X 0,Y 538.045,Z 366.963,A -85,B 0,C 180,E1 -3896.366,E2 -3896.366} C_VEL
LIN {X 0,Y 538.051,Z 366.96,A -85,B 0,C 180,E1 -3898.938,E2 -3898.938} C_VEL
LIN {X 0,Y 538.022,Z 366.962,A -85,B 0,C 180,E1 -3901.89,E2 -3901.89} C_VEL
LIN {X 0,Y 538.027,Z 366.962,A -85,B 0,C 180,E1 -3904.621,E2 -3904.621} C_VEL
LIN {X 0,Y 538.002,Z 366.968,A -85,B 0,C 180,E1 -3907.17,E2 -3907.17} C_VEL
LIN {X 0,Y 538.048,Z 366.956,A -85,B 0,C 180,E1 -3909.794,E2 -3909.794} C_VEL
LIN {X 0,Y 538.012,Z 366.961,A -85,B 0,C 180,E1 -3912.786,E2 -3912.786} C_VEL
LIN {X 0,Y 538.026,Z 366.964,A -85,B 0,C 180,E1 -3915.141,E2 -3915.141} C_VEL
LIN {X 0,Y 538.034,Z 366.963,A -85,B 0,C 180,E1 -3918.228,E2 -3918.228} C_VEL
LIN {X 0,Y 538.009,Z 366.965,A -85,B 0,C 180,E1 -3921.17,E2 -3921.17} C_VEL
LIN {X 0,Y 538.022,Z 366.963,A -85,B 0,C 180,E1 -3924.083,E2 -3924.083} C_VEL
LIN {X 0,Y 538.029,Z 366.968,A -85,B 0,C 180,E1 -3926.728,E2 -3926.728} C_VEL
LIN {X 0,Y 538.031,Z 366.96,A -85,B 0,C 180,E1 -3929.554,E2 -3929.554} C_VEL
LIN {X 0,Y 538.041,Z 366.957,A -85,B 0,C 180,E1 -3931.951,E2 -3931.951} C_VEL
LIN {X 0,Y 538.069,Z 366.96,A -85,B 0,C 180,E1 -3934.468,E2 -3934.468} C_VEL
LIN {X 0,Y 538.016,Z 366.965,A -85,B 0,C 180,E1 -3936.929,E2 -3936.929} C_VEL
LIN {X 0,Y 538.072,Z 366.956,A -85,B 0,C 180,E1 -3940.148,E2 -3940.148} C_VEL
LIN {X 0,Y 538.021,Z 366.961,A -85,B 0,C 180,E1 -3943.299,E2 -3943.299} C_VEL
LIN {X 0,Y 538.057,Z 366.957,A -85,B 0,C 180,E1 -3945.631,E2 -3945.631} C_VEL
LIN {X 0,Y 538.07,Z 366.953,A -85,B 0,C 180,E1 -3948.702,E2 -3948.702} C_VEL
LIN {X 0,Y 538.081,Z 366.951,A -85,B 0,C 180,E1 -3951.74,E2 -3951.74} C_VEL
LIN {X 0,Y 538.159,Z 366.948,A -85,B 0,C 180,E1 -3954.755,E2 -3954.755} C_VEL
LIN {X 0,Y 538.163,Z 366.943,A -85,B 0,C 180,E1 -3957.755,E2 -3957.755} C_VEL
LIN {X 0,Y 538.179,Z 366.941,A -85,B 0,C 180,E1 -3960.749,E2 -3960.749} C_VEL
LIN {X 0,Y 538.137,Z 366.948,A -85,B 0,C 180,E1 -3962.995,E2 -3962.995} C_VEL
LIN {X 0,Y 538.12,Z 366.954,A -85,B 0,C 180,E1 -3965.998,E2 -3965.998} C_VEL
LIN {X 0,Y 538.067,Z 366.947,A -85,B 0,C 180,E1 -3969.018,E2 -3969.018} C_VEL
LIN {X 0,Y 538.078,Z 366.957,A -85,B 0,C 180,E1 -3972.063,E2 -3972.063} C_VEL
LIN {X 0,Y 538.041,Z 366.958,A -85,B 0,C 180,E1 -3975.144,E2 -3975.144} C_VEL
LIN {X 0,Y 538.031,Z 366.961,A -85,B 0,C 180,E1 -3978.271,E2 -3978.271} C_VEL
LIN {X 0,Y 538.038,Z 366.961,A -85,B 0,C 180,E1 -3980.652,E2 -3980.652} C_VEL
LIN {X 0,Y 538.02,Z 366.966,A -85,B 0,C 180,E1 -3983.888,E2 -3983.888} C_VEL
LIN {X 0,Y 538.046,Z 366.959,A -85,B 0,C 180,E1 -3986.367,E2 -3986.367} C_VEL
LIN {X 0,Y 538.053,Z 366.957,A -85,B 0,C 180,E1 -3988.939,E2 -3988.939} C_VEL
LIN {X 0,Y 538.025,Z 366.967,A -85,B 0,C 180,E1 -3991.891,E2 -3991.891} C_VEL
LIN {X 0,Y 538.031,Z 366.96,A -85,B 0,C 180,E1 -3994.622,E2 -3994.622} C_VEL
LIN {X 0,Y 538.005,Z 366.964,A -85,B 0,C 180,E1 -3997.171,E2 -3997.171} C_VEL
LIN {X 0,Y 538.052,Z 366.961,A -85,B 0,C 180,E1 -3999.795,E2 -3999.795} C_VEL
LIN {X 0,Y 538.022,Z 366.962,A -85,B 0,C 180,E1 -4002.786,E2 -4002.786} C_VEL
LIN {X 0,Y 538.028,Z 366.968,A -85,B 0,C 180,E1 -4005.926,E2 -4005.926} C_VEL
LIN {X 0,Y 538.051,Z 366.953,A -85,B 0,C 180,E1 -4009.253,E2 -4009.253} C_VEL
LIN {X 0,Y 537.994,Z 366.972,A -85,B 0,C 180,E1 -4012.123,E2 -4012.123} C_VEL
LIN {X 0,Y 538.021,Z 366.961,A -85,B 0,C 180,E1 -4014.918,E2 -4014.918} C_VEL
LIN {X 0,Y 538.027,Z 366.965,A -85,B 0,C 180,E1 -4017.619,E2 -4017.619} C_VEL
LIN {X 0,Y 538.045,Z 366.966,A -85,B 0,C 180,E1 -4020.241,E2 -4020.241} C_VEL
LIN {X 0,Y 538.068,Z 366.96,A -85,B 0,C 180,E1 -4022.797,E2 -4022.797} C_VEL
LIN {X 0,Y 538.107,Z 367.083,A -85,B 0,C 180,E1 -4024.314,E2 -4024.314} C_VEL
LIN {X 0,Y 539.11,Z 373.515,A -85,B 0,C 180,E1 -4025.662,E2 -4025.662} C_VEL
LIN {X 0,Y 538.76,Z 388.503,A -85,B 0,C 180,E1 -4028.577,E2 -4028.577} C_VEL
LIN {X 0,Y 538.491,Z 405.24,A -85,B 0,C 180,E1 -4031.746,E2 -4031.746} C_VEL
LIN {X 0,Y 538.198,Z 421.921,A -85,B 0,C 180,E1 -4034.861,E2 -4034.861} C_VEL
LIN {X 0,Y 538.14,Z 424.211,A -85,B 0,C 180,E1 -4035.238,E2 -4035.238} C_VEL
LIN {X 0,Y 539.676,Z 434.159,A -85,B 0,C 180,E1 -4035.44,E2 -4035.44} C_VEL
LIN {X 0,Y 539.359,Z 529.002,A -85,B 0,C 180,E1 -4036.723,E2 -4036.723} C_VEL
LIN {X 0,Y 539.199,Z 538.916,A -85,B 0,C 180,E1 -4036.935,E2 -4036.935} C_VEL
LIN {X 0,Y 539.084,Z 548.906,A -85,B 0,C 180,E1 -4037.244,E2 -4037.244} C_VEL
LIN {X 0,Y 538.899,Z 559.266,A -85,B 0,C 180,E1 -4037.67,E2 -4037.67} C_VEL
LIN {X 0,Y 538.716,Z 568.228,A -85,B 0,C 180,E1 -4038.132,E2 -4038.132} C_VEL
LIN {X 0,Y 538.585,Z 577.423,A -85,B 0,C 180,E1 -4038.713,E2 -4038.713} C_VEL
LIN {X 0,Y 538.378,Z 586.153,A -85,B 0,C 180,E1 -4039.375,E2 -4039.375} C_VEL
LIN {X 0,Y 538.212,Z 593.57,A -85,B 0,C 180,E1 -4040.037,E2 -4040.037} C_VEL
LIN {X 0,Y 537.982,Z 602.336,A -85,B 0,C 180,E1 -4040.981,E2 -4040.981} C_VEL
LIN {X 0,Y 537.88,Z 608.301,A -85,B 0,C 180,E1 -4041.737,E2 -4041.737} C_VEL
LIN {X 0,Y 537.754,Z 614.582,A -85,B 0,C 180,E1 -4042.68,E2 -4042.68} C_VEL
LIN {X 0,Y 537.635,Z 620.108,A -85,B 0,C 180,E1 -4043.68,E2 -4043.68} C_VEL
LIN {X 0,Y 537.587,Z 624.888,A -85,B 0,C 180,E1 -4044.75,E2 -4044.75} C_VEL
LIN {X 0,Y 537.603,Z 628.825,A -85,B 0,C 180,E1 -4045.877,E2 -4045.877} C_VEL
LIN {X 0,Y 537.551,Z 631.736,A -85,B 0,C 180,E1 -4047.003,E2 -4047.003} C_VEL
LIN {X 0,Y 537.489,Z 633.215,A -85,B 0,C 180,E1 -4047.752,E2 -4047.752} C_VEL
LIN {X 0,Y 537.442,Z 634.731,A -85,B 0,C 180,E1 -4049.251,E2 -4049.251} C_VEL
LIN {X 0,Y 537.442,Z 635,A -85,B 0,C 180,E1 -4050,E2 -4050} C_VEL
LIN {X 0,Y 537.451,Z 634.142,A -85,B 0,C 180,E1 -4051.499,E2 -4051.499} C_VEL
LIN {X 0,Y 537.489,Z 633.214,A -85,B 0,C 180,E1 -4052.248,E2 -4052.248} C_VEL
LIN {X 0,Y 537.591,Z 629.904,A -85,B 0,C 180,E1 -4053.748,E2 -4053.748} C_VEL
LIN {X 0,Y 537.54,Z 626.305,A -85,B 0,C 180,E1 -4054.875,E2 -4054.875} C_VEL
LIN {X 0,Y 537.673,Z 623.382,A -85,B 0,C 180,E1 -4055.626,E2 -4055.626} C_VEL
LIN {X 0,Y 537.717,Z 617.841,A -85,B 0,C 180,E1 -4056.756,E2 -4056.756} C_VEL
LIN {X 0,Y 537.816,Z 612.216,A -85,B 0,C 180,E1 -4057.698,E2 -4057.698} C_VEL
LIN {X 0,Y 537.964,Z 605.442,A -85,B 0,C 180,E1 -4058.641,E2 -4058.641} C_VEL
LIN {X 0,Y 538.142,Z 597.255,A -85,B 0,C 180,E1 -4059.585,E2 -4059.585} C_VEL
LIN {X 0,Y 538.257,Z 589.444,A -85,B 0,C 180,E1 -4060.343,E2 -4060.343} C_VEL
LIN {X 0,Y 538.486,Z 581.357,A -85,B 0,C 180,E1 -4061.004,E2 -4061.004} C_VEL
LIN {X 0,Y 538.686,Z 571.925,A -85,B 0,C 180,E1 -4061.647,E2 -4061.647} C_VEL
LIN {X 0,Y 538.836,Z 563.195,A -85,B 0,C 180,E1 -4062.141,E2 -4062.141} C_VEL
LIN {X 0,Y 538.994,Z 552.682,A -85,B 0,C 180,E1 -4062.615,E2 -4062.615} C_VEL
LIN {X 0,Y 539.199,Z 542.345,A -85,B 0,C 180,E1 -4062.97,E2 -4062.97} C_VEL
LIN {X 0,Y 539.306,Z 531.619,A -85,B 0,C 180,E1 -4063.23,E2 -4063.23} C_VEL
LIN {X 0,Y 539.486,Z 508.842,A -85,B 0,C 180,E1 -4063.562,E2 -4063.562} C_VEL
LIN {X 0,Y 539.635,Z 432.962,A -85,B 0,C 180,E1 -4064.577,E2 -4064.577} C_VEL
LIN {X 0,Y 538.141,Z 424.202,A -85,B 0,C 180,E1 -4064.762,E2 -4064.762} C_VEL
LIN {X 0,Y 538.242,Z 418.812,A -85,B 0,C 180,E1 -4065.72,E2 -4065.72} C_VEL
LIN {X 0,Y 538.453,Z 403.145,A -85,B 0,C 180,E1 -4068.65,E2 -4068.65} C_VEL
LIN {X 0,Y 538.752,Z 388.522,A -85,B 0,C 180,E1 -4071.423,E2 -4071.423} C_VEL
LIN {X 0,Y 539.086,Z 373.538,A -85,B 0,C 180,E1 -4074.34,E2 -4074.34} C_VEL
LIN {X 0,Y 538.082,Z 367.069,A -85,B 0,C 180,E1 -4075.68,E2 -4075.68} C_VEL
LIN {X 0,Y 538.05,Z 366.965,A -85,B 0,C 180,E1 -4078.049,E2 -4078.049} C_VEL
LIN {X 0,Y 538.032,Z 366.965,A -85,B 0,C 180,E1 -4080.626,E2 -4080.626} C_VEL
LIN {X 0,Y 538.048,Z 366.958,A -85,B 0,C 180,E1 -4083.282,E2 -4083.282} C_VEL
LIN {X 0,Y 538.03,Z 366.965,A -85,B 0,C 180,E1 -4086.002,E2 -4086.002} C_VEL
LIN {X 0,Y 538.018,Z 366.962,A -85,B 0,C 180,E1 -4088.83,E2 -4088.83} C_VEL
LIN {X 0,Y 538.042,Z 366.959,A -85,B 0,C 180,E1 -4091.772,E2 -4091.772} C_VEL
LIN {X 0,Y 538.033,Z 366.96,A -85,B 0,C 180,E1 -4094.859,E2 -4094.859} C_VEL
LIN {X 0,Y 538.039,Z 366.966,A -85,B 0,C 180,E1 -4098.12,E2 -4098.12} C_VEL
LIN {X 0,Y 538.06,Z 366.958,A -85,B 0,C 180,E1 -4100.411,E2 -4100.411} C_VEL
LIN {X 0,Y 538.028,Z 366.961,A -85,B 0,C 180,E1 -4103.067,E2 -4103.067} C_VEL
LIN {X 0,Y 538.025,Z 366.965,A -85,B 0,C 180,E1 -4105.827,E2 -4105.827} C_VEL
LIN {X 0,Y 538.025,Z 366.962,A -85,B 0,C 180,E1 -4108.499,E2 -4108.499} C_VEL
LIN {X 0,Y 538.059,Z 366.956,A -85,B 0,C 180,E1 -4111.099,E2 -4111.099} C_VEL
LIN {X 0,Y 538.042,Z 366.96,A -85,B 0,C 180,E1 -4113.633,E2 -4113.633} C_VEL
LIN {X 0,Y 538.022,Z 366.966,A -85,B 0,C 180,E1 -4116.118,E2 -4116.118} C_VEL
LIN {X 0,Y 538.038,Z 366.961,A -85,B 0,C 180,E1 -4119.348,E2 -4119.348} C_VEL
LIN {X 0,Y 538.053,Z 366.953,A -85,B 0,C 180,E1 -4122.517,E2 -4122.517} C_VEL
LIN {X 0,Y 538.062,Z 366.963,A -85,B 0,C 180,E1 -4125.63,E2 -4125.63} C_VEL
LIN {X 0,Y 538.075,Z 366.951,A -85,B 0,C 180,E1 -4128.701,E2 -4128.701} C_VEL
LIN {X 0,Y 538.085,Z 366.955,A -85,B 0,C 180,E1 -4131.739,E2 -4131.739} C_VEL
LIN {X 0,Y 538.161,Z 366.944,A -85,B 0,C 180,E1 -4134.755,E2 -4134.755} C_VEL
LIN {X 0,Y 538.165,Z 366.948,A -85,B 0,C 180,E1 -4137.754,E2 -4137.754} C_VEL
LIN {X 0,Y 538.182,Z 366.933,A -85,B 0,C 180,E1 -4140.748,E2 -4140.748} C_VEL
LIN {X 0,Y 538.139,Z 366.945,A -85,B 0,C 180,E1 -4142.994,E2 -4142.994} C_VEL
LIN {X 0,Y 538.121,Z 366.952,A -85,B 0,C 180,E1 -4145.997,E2 -4145.997} C_VEL
LIN {X 0,Y 538.068,Z 366.953,A -85,B 0,C 180,E1 -4149.017,E2 -4149.017} C_VEL
LIN {X 0,Y 538.08,Z 366.955,A -85,B 0,C 180,E1 -4152.062,E2 -4152.062} C_VEL
LIN {X 0,Y 538.042,Z 366.962,A -85,B 0,C 180,E1 -4155.143,E2 -4155.143} C_VEL
LIN {X 0,Y 538.028,Z 366.955,A -85,B 0,C 180,E1 -4158.27,E2 -4158.27} C_VEL
LIN {X 0,Y 538.036,Z 366.956,A -85,B 0,C 180,E1 -4160.651,E2 -4160.651} C_VEL
LIN {X 0,Y 538.02,Z 366.965,A -85,B 0,C 180,E1 -4163.887,E2 -4163.887} C_VEL
LIN {X 0,Y 538.046,Z 366.955,A -85,B 0,C 180,E1 -4166.366,E2 -4166.366} C_VEL
LIN {X 0,Y 538.027,Z 366.96,A -85,B 0,C 180,E1 -4168.933,E2 -4168.933} C_VEL
LIN {X 0,Y 538.024,Z 366.964,A -85,B 0,C 180,E1 -4171.89,E2 -4171.89} C_VEL
LIN {X 0,Y 538.027,Z 366.957,A -85,B 0,C 180,E1 -4174.62,E2 -4174.62} C_VEL
LIN {X 0,Y 538.004,Z 366.969,A -85,B 0,C 180,E1 -4177.17,E2 -4177.17} C_VEL
LIN {X 0,Y 538.018,Z 366.959,A -85,B 0,C 180,E1 -4180.269,E2 -4180.269} C_VEL
LIN {X 0,Y 537.368,Z 367.043,A -85,B 0,C 180,E1 -4180.895,E2 -4180.895} C_VEL
LIN {X 0,Y 534.519,Z 367.405,A -85,B 0,C 180,E1 -4181.91,E2 -4181.91} C_VEL
LIN {X 0,Y 532.096,Z 367.711,A -85,B 0,C 180,E1 -4182.727,E2 -4182.727} C_VEL
LIN {X 0,Y 531.048,Z 367.839,A -85,B 0,C 180,E1 -4183.358,E2 -4183.358} C_VEL
LIN {X 0,Y 530.959,Z 367.847,A -85,B 0,C 180,E1 -4183.571,E2 -4183.571} C_VEL
LIN {X 0,Y 530.96,Z 367.836,A -85,B 0,C 180,E1 -4186.505,E2 -4186.505} C_VEL
LIN {X 0,Y 531.022,Z 367.837,A -85,B 0,C 180,E1 -4189.571,E2 -4189.571} C_VEL
LIN {X 0,Y 530.965,Z 367.842,A -85,B 0,C 180,E1 -4192.577,E2 -4192.577} C_VEL
LIN {X 0,Y 530.998,Z 367.836,A -85,B 0,C 180,E1 -4195.311,E2 -4195.311} C_VEL
LIN {X 0,Y 530.979,Z 367.84,A -85,B 0,C 180,E1 -4198.033,E2 -4198.033} C_VEL
LIN {X 0,Y 531.004,Z 367.836,A -85,B 0,C 180,E1 -4200.87,E2 -4200.87} C_VEL
LIN {X 0,Y 531.003,Z 367.845,A -85,B 0,C 180,E1 -4203.256,E2 -4203.256} C_VEL
LIN {X 0,Y 530.994,Z 367.839,A -85,B 0,C 180,E1 -4205.957,E2 -4205.957} C_VEL
LIN {X 0,Y 530.997,Z 367.846,A -85,B 0,C 180,E1 -4209.062,E2 -4209.062} C_VEL
LIN {X 0,Y 531.014,Z 367.836,A -85,B 0,C 180,E1 -4212.278,E2 -4212.278} C_VEL
LIN {X 0,Y 531.016,Z 367.84,A -85,B 0,C 180,E1 -4215.436,E2 -4215.436} C_VEL
LIN {X 0,Y 531.034,Z 367.836,A -85,B 0,C 180,E1 -4218.55,E2 -4218.55} C_VEL
LIN {X 0,Y 531.052,Z 367.834,A -85,B 0,C 180,E1 -4221.629,E2 -4221.629} C_VEL
LIN {X 0,Y 531.122,Z 367.827,A -85,B 0,C 180,E1 -4224.685,E2 -4224.685} C_VEL
LIN {X 0,Y 531.138,Z 367.822,A -85,B 0,C 180,E1 -4227.725,E2 -4227.725} C_VEL
LIN {X 0,Y 531.15,Z 367.825,A -85,B 0,C 180,E1 -4230.758,E2 -4230.758} C_VEL
LIN {X 0,Y 531.102,Z 367.833,A -85,B 0,C 180,E1 -4233.034,E2 -4233.034} C_VEL
LIN {X 0,Y 531.089,Z 367.827,A -85,B 0,C 180,E1 -4236.077,E2 -4236.077} C_VEL
LIN {X 0,Y 531.028,Z 367.841,A -85,B 0,C 180,E1 -4239.138,E2 -4239.138} C_VEL
LIN {X 0,Y 531.037,Z 367.835,A -85,B 0,C 180,E1 -4242.225,E2 -4242.225} C_VEL
LIN {X 0,Y 530.992,Z 367.842,A -85,B 0,C 180,E1 -4245.349,E2 -4245.349} C_VEL
LIN {X 0,Y 531.012,Z 367.837,A -85,B 0,C 180,E1 -4247.722,E2 -4247.722} C_VEL
LIN {X 0,Y 530.995,Z 367.846,A -85,B 0,C 180,E1 -4250.938,E2 -4250.938} C_VEL
LIN {X 0,Y 530.975,Z 367.842,A -85,B 0,C 180,E1 -4254.224,E2 -4254.224} C_VEL
LIN {X 0,Y 531.007,Z 367.845,A -85,B 0,C 180,E1 -4256.743,E2 -4256.743} C_VEL
LIN {X 0,Y 530.995,Z 367.835,A -85,B 0,C 180,E1 -4259.321,E2 -4259.321} C_VEL
LIN {X 0,Y 530.974,Z 367.841,A -85,B 0,C 180,E1 -4262.103,E2 -4262.103} C_VEL
LIN {X 0,Y 530.984,Z 367.839,A -85,B 0,C 180,E1 -4264.854,E2 -4264.854} C_VEL
LIN {X 0,Y 530.96,Z 367.842,A -85,B 0,C 180,E1 -4267.507,E2 -4267.507} C_VEL
LIN {X 0,Y 531.02,Z 367.837,A -85,B 0,C 180,E1 -4270.428,E2 -4270.428} C_VEL
LIN {X 0,Y 530.958,Z 367.836,A -85,B 0,C 180,E1 -4273.494,E2 -4273.494} C_VEL
LIN {X 0,Y 530.961,Z 367.848,A -85,B 0,C 180,E1 -4276.506,E2 -4276.506} C_VEL
LIN {X 0,Y 530.978,Z 367.836,A -85,B 0,C 180,E1 -4279.567,E2 -4279.567} C_VEL
LIN {X 0,Y 530.969,Z 367.849,A -85,B 0,C 180,E1 -4282.576,E2 -4282.576} C_VEL
LIN {X 0,Y 530.996,Z 367.832,A -85,B 0,C 180,E1 -4285.311,E2 -4285.311} C_VEL
LIN {X 0,Y 530.976,Z 367.841,A -85,B 0,C 180,E1 -4288.033,E2 -4288.033} C_VEL
LIN {X 0,Y 531,Z 367.837,A -85,B 0,C 180,E1 -4290.87,E2 -4290.87} C_VEL
LIN {X 0,Y 531.005,Z 367.832,A -85,B 0,C 180,E1 -4293.257,E2 -4293.257} C_VEL
LIN {X 0,Y 530.99,Z 367.839,A -85,B 0,C 180,E1 -4295.958,E2 -4295.958} C_VEL
LIN {X 0,Y 530.995,Z 367.834,A -85,B 0,C 180,E1 -4299.062,E2 -4299.062} C_VEL
LIN {X 0,Y 531.009,Z 367.835,A -85,B 0,C 180,E1 -4302.278,E2 -4302.278} C_VEL
LIN {X 0,Y 531.012,Z 367.835,A -85,B 0,C 180,E1 -4305.436,E2 -4305.436} C_VEL
LIN {X 0,Y 531.042,Z 367.831,A -85,B 0,C 180,E1 -4308.55,E2 -4308.55} C_VEL
LIN {X 0,Y 531.051,Z 367.825,A -85,B 0,C 180,E1 -4311.63,E2 -4311.63} C_VEL
LIN {X 0,Y 531.117,Z 367.826,A -85,B 0,C 180,E1 -4314.686,E2 -4314.686} C_VEL
LIN {X 0,Y 531.135,Z 367.818,A -85,B 0,C 180,E1 -4317.725,E2 -4317.725} C_VEL
LIN {X 0,Y 531.149,Z 367.817,A -85,B 0,C 180,E1 -4320.759,E2 -4320.759} C_VEL
LIN {X 0,Y 531.103,Z 367.824,A -85,B 0,C 180,E1 -4323.035,E2 -4323.035} C_VEL
LIN {X 0,Y 531.079,Z 367.832,A -85,B 0,C 180,E1 -4326.078,E2 -4326.078} C_VEL
LIN {X 0,Y 531.027,Z 367.823,A -85,B 0,C 180,E1 -4329.139,E2 -4329.139} C_VEL
LIN {X 0,Y 531.035,Z 367.837,A -85,B 0,C 180,E1 -4332.225,E2 -4332.225} C_VEL
LIN {X 0,Y 530.991,Z 367.836,A -85,B 0,C 180,E1 -4335.35,E2 -4335.35} C_VEL
LIN {X 0,Y 531.012,Z 367.832,A -85,B 0,C 180,E1 -4337.723,E2 -4337.723} C_VEL
LIN {X 0,Y 530.998,Z 367.835,A -85,B 0,C 180,E1 -4340.938,E2 -4340.938} C_VEL
LIN {X 0,Y 530.976,Z 367.845,A -85,B 0,C 180,E1 -4344.225,E2 -4344.225} C_VEL
LIN {X 0,Y 531.008,Z 367.831,A -85,B 0,C 180,E1 -4346.744,E2 -4346.744} C_VEL
LIN {X 0,Y 530.997,Z 367.836,A -85,B 0,C 180,E1 -4349.322,E2 -4349.322} C_VEL
LIN {X 0,Y 530.978,Z 367.846,A -85,B 0,C 180,E1 -4352.104,E2 -4352.104} C_VEL
LIN {X 0,Y 530.987,Z 367.836,A -85,B 0,C 180,E1 -4354.855,E2 -4354.855} C_VEL
LIN {X 0,Y 530.964,Z 367.843,A -85,B 0,C 180,E1 -4357.508,E2 -4357.508} C_VEL
LIN {X 0,Y 531.024,Z 367.836,A -85,B 0,C 180,E1 -4360.429,E2 -4360.429} C_VEL
LIN {X 0,Y 530.964,Z 367.843,A -85,B 0,C 180,E1 -4363.495,E2 -4363.495} C_VEL
LIN {X 0,Y 530.963,Z 367.844,A -85,B 0,C 180,E1 -4366.506,E2 -4366.506} C_VEL
LIN {X 0,Y 530.988,Z 367.832,A -85,B 0,C 180,E1 -4368.976,E2 -4368.976} C_VEL
LIN {X 0,Y 530.959,Z 367.844,A -85,B 0,C 180,E1 -4371.53,E2 -4371.53} C_VEL
LIN {X 0,Y 530.983,Z 367.842,A -85,B 0,C 180,E1 -4374.383,E2 -4374.383} C_VEL
LIN {X 0,Y 530.971,Z 367.839,A -85,B 0,C 180,E1 -4377.134,E2 -4377.134} C_VEL
LIN {X 0,Y 530.988,Z 367.844,A -85,B 0,C 180,E1 -4379.805,E2 -4379.805} C_VEL
LIN {X 0,Y 531.018,Z 367.841,A -85,B 0,C 180,E1 -4382.467,E2 -4382.467} C_VEL
LIN {X 0,Y 531.05,Z 367.969,A -85,B 0,C 180,E1 -4384.149,E2 -4384.149} C_VEL
LIN {X 0,Y 532.126,Z 375.25,A -85,B 0,C 180,E1 -4385.688,E2 -4385.688} C_VEL
LIN {X 0,Y 531.771,Z 389.421,A -85,B 0,C 180,E1 -4388.485,E2 -4388.485} C_VEL
LIN {X 0,Y 531.498,Z 405.105,A -85,B 0,C 180,E1 -4391.498,E2 -4391.498} C_VEL
LIN {X 0,Y 531.151,Z 422.902,A -85,B 0,C 180,E1 -4394.876,E2 -4394.876} C_VEL
LIN {X 0,Y 531.152,Z 424.308,A -85,B 0,C 180,E1 -4395.057,E2 -4395.057} C_VEL
LIN {X 0,Y 532.805,Z 434.104,A -85,B 0,C 180,E1 -4395.25,E2 -4395.25} C_VEL
LIN {X 0,Y 532.447,Z 528.806,A -85,B 0,C 180,E1 -4396.548,E2 -4396.548} C_VEL
LIN {X 0,Y 532.298,Z 538.721,A -85,B 0,C 180,E1 -4396.763,E2 -4396.763} C_VEL
LIN {X 0,Y 532.148,Z 548.71,A -85,B 0,C 180,E1 -4397.074,E2 -4397.074} C_VEL
LIN {X 0,Y 531.943,Z 559.07,A -85,B 0,C 180,E1 -4397.506,E2 -4397.506} C_VEL
LIN {X 0,Y 531.733,Z 568.969,A -85,B 0,C 180,E1 -4398.031,E2 -4398.031} C_VEL
LIN {X 0,Y 531.584,Z 577.227,A -85,B 0,C 180,E1 -4398.562,E2 -4398.562} C_VEL
LIN {X 0,Y 531.369,Z 585.957,A -85,B 0,C 180,E1 -4399.233,E2 -4399.233} C_VEL
LIN {X 0,Y 531.186,Z 593.382,A -85,B 0,C 180,E1 -4399.904,E2 -4399.904} C_VEL
LIN {X 0,Y 530.936,Z 602.179,A -85,B 0,C 180,E1 -4400.861,E2 -4400.861} C_VEL
LIN {X 0,Y 530.812,Z 608.17,A -85,B 0,C 180,E1 -4401.626,E2 -4401.626} C_VEL
LIN {X 0,Y 530.681,Z 614.481,A -85,B 0,C 180,E1 -4402.581,E2 -4402.581} C_VEL
LIN {X 0,Y 530.545,Z 620.509,A -85,B 0,C 180,E1 -4403.697,E2 -4403.697} C_VEL
LIN {X 0,Y 530.524,Z 624.842,A -85,B 0,C 180,E1 -4404.68,E2 -4404.68} C_VEL
LIN {X 0,Y 530.523,Z 628.802,A -85,B 0,C 180,E1 -4405.822,E2 -4405.822} C_VEL
LIN {X 0,Y 530.457,Z 631.726,A -85,B 0,C 180,E1 -4406.962,E2 -4406.962} C_VEL
LIN {X 0,Y 530.411,Z 633.216,A -85,B 0,C 180,E1 -4407.722,E2 -4407.722} C_VEL
LIN {X 0,Y 530.344,Z 634.723,A -85,B 0,C 180,E1 -4409.241,E2 -4409.241} C_VEL
LIN {X 0,Y 530.342,Z 635,A -85,B 0,C 180,E1 -4410,E2 -4410} C_VEL
LIN {X 0,Y 530.361,Z 634.134,A -85,B 0,C 180,E1 -4411.519,E2 -4411.519} C_VEL
LIN {X 0,Y 530.411,Z 633.215,A -85,B 0,C 180,E1 -4412.278,E2 -4412.278} C_VEL
LIN {X 0,Y 530.516,Z 629.887,A -85,B 0,C 180,E1 -4413.798,E2 -4413.798} C_VEL
LIN {X 0,Y 530.459,Z 626.265,A -85,B 0,C 180,E1 -4414.94,E2 -4414.94} C_VEL
LIN {X 0,Y 530.606,Z 623.329,A -85,B 0,C 180,E1 -4415.701,E2 -4415.701} C_VEL
LIN {X 0,Y 530.643,Z 617.755,A -85,B 0,C 180,E1 -4416.846,E2 -4416.846} C_VEL
LIN {X 0,Y 530.737,Z 612.103,A -85,B 0,C 180,E1 -4417.801,E2 -4417.801} C_VEL
LIN {X 0,Y 530.888,Z 605.298,A -85,B 0,C 180,E1 -4418.757,E2 -4418.757} C_VEL
LIN {X 0,Y 531.092,Z 597.079,A -85,B 0,C 180,E1 -4419.714,E2 -4419.714} C_VEL
LIN {X 0,Y 531.274,Z 589.249,A -85,B 0,C 180,E1 -4420.48,E2 -4420.48} C_VEL
LIN {X 0,Y 531.473,Z 581.161,A -85,B 0,C 180,E1 -4421.151,E2 -4421.151} C_VEL
LIN {X 0,Y 531.734,Z 571.031,A -85,B 0,C 180,E1 -4421.844,E2 -4421.844} C_VEL
LIN {X 0,Y 531.88,Z 562.999,A -85,B 0,C 180,E1 -4422.302,E2 -4422.302} C_VEL
LIN {X 0,Y 532.081,Z 552.487,A -85,B 0,C 180,E1 -4422.782,E2 -4422.782} C_VEL
LIN {X 0,Y 532.261,Z 542.15,A -85,B 0,C 180,E1 -4423.142,E2 -4423.142} C_VEL
LIN {X 0,Y 532.411,Z 531.425,A -85,B 0,C 180,E1 -4423.405,E2 -4423.405} C_VEL
LIN {X 0,Y 532.575,Z 508.647,A -85,B 0,C 180,E1 -4423.741,E2 -4423.741} C_VEL
LIN {X 0,Y 532.724,Z 433.508,A -85,B 0,C 180,E1 -4424.76,E2 -4424.76} C_VEL
LIN {X 0,Y 531.153,Z 424.298,A -85,B 0,C 180,E1 -4424.943,E2 -4424.943} C_VEL
LIN {X 0,Y 531.152,Z 422.899,A -85,B 0,C 180,E1 -4425.125,E2 -4425.125} C_VEL
LIN {X 0,Y 531.499,Z 405.102,A -85,B 0,C 180,E1 -4428.503,E2 -4428.503} C_VEL
LIN {X 0,Y 531.767,Z 389.418,A -85,B 0,C 180,E1 -4431.515,E2 -4431.515} C_VEL
LIN {X 0,Y 532.114,Z 375.279,A -85,B 0,C 180,E1 -4434.309,E2 -4434.309} C_VEL
LIN {X 0,Y 531.227,Z 368.883,A -85,B 0,C 180,E1 -4435.639,E2 -4435.639} C_VEL
LIN {X 0,Y 531.026,Z 367.923,A -85,B 0,C 180,E1 -4435.896,E2 -4435.896} C_VEL
LIN {X 0,Y 531.003,Z 367.843,A -85,B 0,C 180,E1 -4438.455,E2 -4438.455} C_VEL
LIN {X 0,Y 530.964,Z 367.843,A -85,B 0,C 180,E1 -4441.079,E2 -4441.079} C_VEL
LIN {X 0,Y 530.994,Z 367.842,A -85,B 0,C 180,E1 -4443.772,E2 -4443.772} C_VEL
LIN {X 0,Y 530.971,Z 367.842,A -85,B 0,C 180,E1 -4446.557,E2 -4446.557} C_VEL
LIN {X 0,Y 530.986,Z 367.842,A -85,B 0,C 180,E1 -4449.854,E2 -4449.854} C_VEL
LIN {X 0,Y 530.982,Z 367.841,A -85,B 0,C 180,E1 -4452.456,E2 -4452.456} C_VEL
LIN {X 0,Y 530.989,Z 367.841,A -85,B 0,C 180,E1 -4455.62,E2 -4455.62} C_VEL
LIN {X 0,Y 531.008,Z 367.836,A -85,B 0,C 180,E1 -4458.565,E2 -4458.565} C_VEL
LIN {X 0,Y 530.969,Z 367.84,A -85,B 0,C 180,E1 -4461.346,E2 -4461.346} C_VEL
LIN {X 0,Y 530.977,Z 367.839,A -85,B 0,C 180,E1 -4464.381,E2 -4464.381} C_VEL
LIN {X 0,Y 530.972,Z 367.837,A -85,B 0,C 180,E1 -4467.133,E2 -4467.133} C_VEL
LIN {X 0,Y 530.987,Z 367.846,A -85,B 0,C 180,E1 -4469.804,E2 -4469.804} C_VEL
LIN {X 0,Y 531.016,Z 367.83,A -85,B 0,C 180,E1 -4472.466,E2 -4472.466} C_VEL
LIN {X 0,Y 531.005,Z 367.832,A -85,B 0,C 180,E1 -4474.942,E2 -4474.942} C_VEL
LIN {X 0,Y 530.971,Z 367.841,A -85,B 0,C 180,E1 -4478.246,E2 -4478.246} C_VEL
LIN {X 0,Y 530.995,Z 367.83,A -85,B 0,C 180,E1 -4480.677,E2 -4480.677} C_VEL
LIN {X 0,Y 530.986,Z 367.833,A -85,B 0,C 180,E1 -4483.071,E2 -4483.071} C_VEL
LIN {X 0,Y 531.018,Z 367.837,A -85,B 0,C 180,E1 -4485.435,E2 -4485.435} C_VEL
LIN {X 0,Y 531.035,Z 367.828,A -85,B 0,C 180,E1 -4488.549,E2 -4488.549} C_VEL
LIN {X 0,Y 531.055,Z 367.827,A -85,B 0,C 180,E1 -4491.629,E2 -4491.629} C_VEL
LIN {X 0,Y 531.12,Z 367.821,A -85,B 0,C 180,E1 -4494.685,E2 -4494.685} C_VEL
LIN {X 0,Y 531.137,Z 367.823,A -85,B 0,C 180,E1 -4497.725,E2 -4497.725} C_VEL
LIN {X 0,Y 531.152,Z 367.808,A -85,B 0,C 180,E1 -4500.758,E2 -4500.758} C_VEL
LIN {X 0,Y 531.105,Z 367.822,A -85,B 0,C 180,E1 -4503.034,E2 -4503.034} C_VEL
LIN {X 0,Y 531.081,Z 367.828,A -85,B 0,C 180,E1 -4506.077,E2 -4506.077} C_VEL
LIN {X 0,Y 531.028,Z 367.831,A -85,B 0,C 180,E1 -4509.138,E2 -4509.138} C_VEL
LIN {X 0,Y 531.038,Z 367.83,A -85,B 0,C 180,E1 -4512.225,E2 -4512.225} C_VEL
LIN {X 0,Y 530.993,Z 367.844,A -85,B 0,C 180,E1 -4515.349,E2 -4515.349} C_VEL
LIN {X 0,Y 530.987,Z 367.831,A -85,B 0,C 180,E1 -4518.521,E2 -4518.521} C_VEL
LIN {X 0,Y 530.996,Z 367.834,A -85,B 0,C 180,E1 -4520.938,E2 -4520.938} C_VEL
LIN {X 0,Y 530.976,Z 367.839,A -85,B 0,C 180,E1 -4524.224,E2 -4524.224} C_VEL
LIN {X 0,Y 531.008,Z 367.832,A -85,B 0,C 180,E1 -4526.743,E2 -4526.743} C_VEL
LIN {X 0,Y 530.978,Z 367.843,A -85,B 0,C 180,E1 -4529.322,E2 -4529.322} C_VEL
LIN {X 0,Y 530.976,Z 367.84,A -85,B 0,C 180,E1 -4532.103,E2 -4532.103} C_VEL
LIN {X 0,Y 530.984,Z 367.835,A -85,B 0,C 180,E1 -4534.854,E2 -4534.854} C_VEL
LIN {X 0,Y 530.963,Z 367.849,A -85,B 0,C 180,E1 -4537.507,E2 -4537.507} C_VEL
LIN {X 0,Y 530.981,Z 367.835,A -85,B 0,C 180,E1 -4540.432,E2 -4540.432} C_VEL
LIN {X 0,Y 530.967,Z 367.849,A -85,B 0,C 180,E1 -4543.282,E2 -4543.282} C_VEL
LIN {X 0,Y 530.959,Z 367.847,A -85,B 0,C 180,E1 -4543.571,E2 -4543.571} C_VEL
LIN {X 0,Y 530.286,Z 367.927,A -85,B 0,C 180,E1 -4544.205,E2 -4544.205} C_VEL
LIN {X 0,Y 527.437,Z 368.286,A -85,B 0,C 180,E1 -4545.234,E2 -4545.234} C_VEL
LIN {X 0,Y 525.033,Z 368.583,A -85,B 0,C 180,E1 -4546.062,E2 -4546.062} C_VEL
LIN {X 0,Y 524,Z 368.706,A -85,B 0,C 180,E1 -4546.702,E2 -4546.702} C_VEL
LIN {X 0,Y 523.915,Z 368.714,A -85,B 0,C 180,E1 -4546.918,E2 -4546.918} C_VEL
LIN {X 0,Y 523.975,Z 368.711,A -85,B 0,C 180,E1 -4549.923,E2 -4549.923} C_VEL
LIN {X 0,Y 523.908,Z 368.724,A -85,B 0,C 180,E1 -4552.868,E2 -4552.868} C_VEL
LIN {X 0,Y 523.941,Z 368.714,A -85,B 0,C 180,E1 -4555.711,E2 -4555.711} C_VEL
LIN {X 0,Y 523.929,Z 368.719,A -85,B 0,C 180,E1 -4558.457,E2 -4558.457} C_VEL
LIN {X 0,Y 523.948,Z 368.716,A -85,B 0,C 180,E1 -4561.126,E2 -4561.126} C_VEL
LIN {X 0,Y 523.981,Z 368.712,A -85,B 0,C 180,E1 -4563.98,E2 -4563.98} C_VEL
LIN {X 0,Y 523.933,Z 368.718,A -85,B 0,C 180,E1 -4566.271,E2 -4566.271} C_VEL
LIN {X 0,Y 523.943,Z 368.721,A -85,B 0,C 180,E1 -4568.767,E2 -4568.767} C_VEL
LIN {X 0,Y 523.951,Z 368.723,A -85,B 0,C 180,E1 -4571.221,E2 -4571.221} C_VEL
LIN {X 0,Y 523.934,Z 368.72,A -85,B 0,C 180,E1 -4573.639,E2 -4573.639} C_VEL
LIN {X 0,Y 523.937,Z 368.718,A -85,B 0,C 180,E1 -4576.028,E2 -4576.028} C_VEL
LIN {X 0,Y 524.009,Z 368.71,A -85,B 0,C 180,E1 -4578.394,E2 -4578.394} C_VEL
LIN {X 0,Y 524,Z 368.714,A -85,B 0,C 180,E1 -4581.516,E2 -4581.516} C_VEL
LIN {X 0,Y 524.083,Z 368.703,A -85,B 0,C 180,E1 -4584.614,E2 -4584.614} C_VEL
LIN {X 0,Y 524.11,Z 368.698,A -85,B 0,C 180,E1 -4587.694,E2 -4587.694} C_VEL
LIN {X 0,Y 524.12,Z 368.701,A -85,B 0,C 180,E1 -4590.768,E2 -4590.768} C_VEL
LIN {X 0,Y 524.069,Z 368.708,A -85,B 0,C 180,E1 -4593.075,E2 -4593.075} C_VEL
LIN {X 0,Y 524.05,Z 368.705,A -85,B 0,C 180,E1 -4596.159,E2 -4596.159} C_VEL
LIN {X 0,Y 523.996,Z 368.715,A -85,B 0,C 180,E1 -4599.262,E2 -4599.262} C_VEL
LIN {X 0,Y 523.999,Z 368.711,A -85,B 0,C 180,E1 -4601.739,E2 -4601.739} C_VEL
LIN {X 0,Y 523.989,Z 368.718,A -85,B 0,C 180,E1 -4605.052,E2 -4605.052} C_VEL
LIN {X 0,Y 523.96,Z 368.715,A -85,B 0,C 180,E1 -4607.969,E2 -4607.969} C_VEL
LIN {X 0,Y 523.967,Z 368.717,A -85,B 0,C 180,E1 -4610.41,E2 -4610.41} C_VEL
LIN {X 0,Y 523.912,Z 368.728,A -85,B 0,C 180,E1 -4612.893,E2 -4612.893} C_VEL
LIN {X 0,Y 523.95,Z 368.717,A -85,B 0,C 180,E1 -4615.418,E2 -4615.418} C_VEL
LIN {X 0,Y 523.966,Z 368.713,A -85,B 0,C 180,E1 -4617.998,E2 -4617.998} C_VEL
LIN {X 0,Y 523.947,Z 368.722,A -85,B 0,C 180,E1 -4620.856,E2 -4620.856} C_VEL
LIN {X 0,Y 523.956,Z 368.71,A -85,B 0,C 180,E1 -4623.735,E2 -4623.735} C_VEL
LIN {X 0,Y 523.917,Z 368.719,A -85,B 0,C 180,E1 -4626.404,E2 -4626.404} C_VEL
LIN {X 0,Y 523.926,Z 368.719,A -85,B 0,C 180,E1 -4629.083,E2 -4629.083} C_VEL
LIN {X 0,Y 523.965,Z 368.701,A -85,B 0,C 180,E1 -4631.312,E2 -4631.312} C_VEL
LIN {X 0,Y 523.949,Z 368.719,A -85,B 0,C 180,E1 -4634.691,E2 -4634.691} C_VEL
LIN {X 0,Y 523.951,Z 368.714,A -85,B 0,C 180,E1 -4637.882,E2 -4637.882} C_VEL
LIN {X 0,Y 523.917,Z 368.724,A -85,B 0,C 180,E1 -4640.916,E2 -4640.916} C_VEL
LIN {X 0,Y 523.921,Z 368.718,A -85,B 0,C 180,E1 -4643.828,E2 -4643.828} C_VEL
LIN {X 0,Y 523.937,Z 368.721,A -85,B 0,C 180,E1 -4646.636,E2 -4646.636} C_VEL
LIN {X 0,Y 523.957,Z 368.714,A -85,B 0,C 180,E1 -4649.356,E2 -4649.356} C_VEL
LIN {X 0,Y 523.973,Z 368.713,A -85,B 0,C 180,E1 -4652.281,E2 -4652.281} C_VEL
LIN {X 0,Y 523.948,Z 368.721,A -85,B 0,C 180,E1 -4654.582,E2 -4654.582} C_VEL
LIN {X 0,Y 523.91,Z 368.721,A -85,B 0,C 180,E1 -4657.107,E2 -4657.107} C_VEL
LIN {X 0,Y 523.972,Z 368.708,A -85,B 0,C 180,E1 -4659.866,E2 -4659.866} C_VEL
LIN {X 0,Y 523.964,Z 368.715,A -85,B 0,C 180,E1 -4662.838,E2 -4662.838} C_VEL
LIN {X 0,Y 523.969,Z 368.713,A -85,B 0,C 180,E1 -4665.236,E2 -4665.236} C_VEL
LIN {X 0,Y 524.008,Z 368.709,A -85,B 0,C 180,E1 -4668.394,E2 -4668.394} C_VEL
LIN {X 0,Y 523.999,Z 368.703,A -85,B 0,C 180,E1 -4671.516,E2 -4671.516} C_VEL
LIN {X 0,Y 524.078,Z 368.704,A -85,B 0,C 180,E1 -4674.614,E2 -4674.614} C_VEL
LIN {X 0,Y 524.107,Z 368.693,A -85,B 0,C 180,E1 -4677.695,E2 -4677.695} C_VEL
LIN {X 0,Y 524.119,Z 368.692,A -85,B 0,C 180,E1 -4680.769,E2 -4680.769} C_VEL
LIN {X 0,Y 524.069,Z 368.7,A -85,B 0,C 180,E1 -4683.075,E2 -4683.075} C_VEL
LIN {X 0,Y 524.041,Z 368.71,A -85,B 0,C 180,E1 -4686.159,E2 -4686.159} C_VEL
LIN {X 0,Y 523.995,Z 368.698,A -85,B 0,C 180,E1 -4689.262,E2 -4689.262} C_VEL
LIN {X 0,Y 523.997,Z 368.706,A -85,B 0,C 180,E1 -4691.74,E2 -4691.74} C_VEL
LIN {X 0,Y 523.987,Z 368.709,A -85,B 0,C 180,E1 -4695.053,E2 -4695.053} C_VEL
LIN {X 0,Y 523.96,Z 368.713,A -85,B 0,C 180,E1 -4697.97,E2 -4697.97} C_VEL
LIN {X 0,Y 523.968,Z 368.717,A -85,B 0,C 180,E1 -4700.411,E2 -4700.411} C_VEL
LIN {X 0,Y 523.913,Z 368.719,A -85,B 0,C 180,E1 -4702.894,E2 -4702.894} C_VEL
LIN {X 0,Y 523.951,Z 368.712,A -85,B 0,C 180,E1 -4705.419,E2 -4705.419} C_VEL
LIN {X 0,Y 523.967,Z 368.713,A -85,B 0,C 180,E1 -4707.999,E2 -4707.999} C_VEL
LIN {X 0,Y 523.949,Z 368.715,A -85,B 0,C 180,E1 -4710.857,E2 -4710.857} C_VEL
LIN {X 0,Y 523.96,Z 368.713,A -85,B 0,C 180,E1 -4713.736,E2 -4713.736} C_VEL
LIN {X 0,Y 523.92,Z 368.723,A -85,B 0,C 180,E1 -4716.405,E2 -4716.405} C_VEL
LIN {X 0,Y 523.929,Z 368.715,A -85,B 0,C 180,E1 -4719.084,E2 -4719.084} C_VEL
LIN {X 0,Y 523.97,Z 368.712,A -85,B 0,C 180,E1 -4721.313,E2 -4721.313} C_VEL
LIN {X 0,Y 523.954,Z 368.715,A -85,B 0,C 180,E1 -4724.692,E2 -4724.692} C_VEL
LIN {X 0,Y 523.955,Z 368.72,A -85,B 0,C 180,E1 -4727.882,E2 -4727.882} C_VEL
LIN {X 0,Y 523.923,Z 368.718,A -85,B 0,C 180,E1 -4730.916,E2 -4730.916} C_VEL
LIN {X 0,Y 523.929,Z 368.721,A -85,B 0,C 180,E1 -4733.828,E2 -4733.828} C_VEL
LIN {X 0,Y 523.943,Z 368.715,A -85,B 0,C 180,E1 -4736.636,E2 -4736.636} C_VEL
LIN {X 0,Y 523.964,Z 368.717,A -85,B 0,C 180,E1 -4739.357,E2 -4739.357} C_VEL
LIN {X 0,Y 523.981,Z 368.718,A -85,B 0,C 180,E1 -4742.281,E2 -4742.281} C_VEL
LIN {X 0,Y 523.995,Z 368.847,A -85,B 0,C 180,E1 -4743.979,E2 -4743.979} C_VEL
LIN {X 0,Y 525.135,Z 375.965,A -85,B 0,C 180,E1 -4745.514,E2 -4745.514} C_VEL
LIN {X 0,Y 524.795,Z 390.323,A -85,B 0,C 180,E1 -4748.391,E2 -4748.391} C_VEL
LIN {X 0,Y 524.467,Z 407.06,A -85,B 0,C 180,E1 -4751.645,E2 -4751.645} C_VEL
LIN {X 0,Y 524.132,Z 423.78,A -85,B 0,C 180,E1 -4754.832,E2 -4754.832} C_VEL
LIN {X 0,Y 525.79,Z 433.865,A -85,B 0,C 180,E1 -4755.048,E2 -4755.048} C_VEL
LIN {X 0,Y 525.552,Z 528.612,A -85,B 0,C 180,E1 -4756.368,E2 -4756.368} C_VEL
LIN {X 0,Y 525.383,Z 538.526,A -85,B 0,C 180,E1 -4756.585,E2 -4756.585} C_VEL
LIN {X 0,Y 525.237,Z 548.515,A -85,B 0,C 180,E1 -4756.901,E2 -4756.901} C_VEL
LIN {X 0,Y 524.983,Z 558.874,A -85,B 0,C 180,E1 -4757.338,E2 -4757.338} C_VEL
LIN {X 0,Y 524.782,Z 568.618,A -85,B 0,C 180,E1 -4757.86,E2 -4757.86} C_VEL
LIN {X 0,Y 524.588,Z 577.031,A -85,B 0,C 180,E1 -4758.407,E2 -4758.407} C_VEL
LIN {X 0,Y 524.369,Z 585.762,A -85,B 0,C 180,E1 -4759.088,E2 -4759.088} C_VEL
LIN {X 0,Y 524.159,Z 593.185,A -85,B 0,C 180,E1 -4759.767,E2 -4759.767} C_VEL
LIN {X 0,Y 523.901,Z 601.983,A -85,B 0,C 180,E1 -4760.737,E2 -4760.737} C_VEL
LIN {X 0,Y 523.77,Z 607.975,A -85,B 0,C 180,E1 -4761.513,E2 -4761.513} C_VEL
LIN {X 0,Y 523.63,Z 614.285,A -85,B 0,C 180,E1 -4762.481,E2 -4762.481} C_VEL
LIN {X 0,Y 523.521,Z 619.435,A -85,B 0,C 180,E1 -4763.422,E2 -4763.422} C_VEL
LIN {X 0,Y 523.462,Z 624.647,A -85,B 0,C 180,E1 -4764.608,E2 -4764.608} C_VEL
LIN {X 0,Y 523.425,Z 628.606,A -85,B 0,C 180,E1 -4765.765,E2 -4765.765} C_VEL
LIN {X 0,Y 523.367,Z 631.533,A -85,B 0,C 180,E1 -4766.921,E2 -4766.921} C_VEL
LIN {X 0,Y 523.334,Z 633.029,A -85,B 0,C 180,E1 -4767.691,E2 -4767.691} C_VEL
LIN {X 0,Y 523.25,Z 634.544,A -85,B 0,C 180,E1 -4769.231,E2 -4769.231} C_VEL
LIN {X 0,Y 523.246,Z 634.822,A -85,B 0,C 180,E1 -4770,E2 -4770} C_VEL
LIN {X 0,Y 523.275,Z 633.951,A -85,B 0,C 180,E1 -4771.539,E2 -4771.539} C_VEL
LIN {X 0,Y 523.335,Z 633.028,A -85,B 0,C 180,E1 -4772.309,E2 -4772.309} C_VEL
LIN {X 0,Y 523.443,Z 629.692,A -85,B 0,C 180,E1 -4773.849,E2 -4773.849} C_VEL
LIN {X 0,Y 523.383,Z 626.07,A -85,B 0,C 180,E1 -4775.007,E2 -4775.007} C_VEL
LIN {X 0,Y 523.517,Z 623.134,A -85,B 0,C 180,E1 -4775.779,E2 -4775.779} C_VEL
LIN {X 0,Y 523.579,Z 617.56,A -85,B 0,C 180,E1 -4776.939,E2 -4776.939} C_VEL
LIN {X 0,Y 523.679,Z 611.907,A -85,B 0,C 180,E1 -4777.907,E2 -4777.907} C_VEL
LIN {X 0,Y 523.822,Z 605.102,A -85,B 0,C 180,E1 -4778.876,E2 -4778.876} C_VEL
LIN {X 0,Y 524.056,Z 596.883,A -85,B 0,C 180,E1 -4779.845,E2 -4779.845} C_VEL
LIN {X 0,Y 524.282,Z 589.053,A -85,B 0,C 180,E1 -4780.621,E2 -4780.621} C_VEL
LIN {X 0,Y 524.495,Z 580.965,A -85,B 0,C 180,E1 -4781.301,E2 -4781.301} C_VEL
LIN {X 0,Y 524.732,Z 571.926,A -85,B 0,C 180,E1 -4781.937,E2 -4781.937} C_VEL
LIN {X 0,Y 524.923,Z 562.804,A -85,B 0,C 180,E1 -4782.468,E2 -4782.468} C_VEL
LIN {X 0,Y 525.164,Z 552.292,A -85,B 0,C 180,E1 -4782.953,E2 -4782.953} C_VEL
LIN {X 0,Y 525.323,Z 541.954,A -85,B 0,C 180,E1 -4783.318,E2 -4783.318} C_VEL
LIN {X 0,Y 525.517,Z 531.23,A -85,B 0,C 180,E1 -4783.584,E2 -4783.584} C_VEL
LIN {X 0,Y 525.698,Z 508.452,A -85,B 0,C 180,E1 -4783.924,E2 -4783.924} C_VEL
LIN {X 0,Y 525.788,Z 433.952,A -85,B 0,C 180,E1 -4784.95,E2 -4784.95} C_VEL
LIN {X 0,Y 524.124,Z 423.854,A -85,B 0,C 180,E1 -4785.162,E2 -4785.162} C_VEL
LIN {X 0,Y 524.138,Z 420.59,A -85,B 0,C 180,E1 -4785.755,E2 -4785.755} C_VEL
LIN {X 0,Y 524.45,Z 404.966,A -85,B 0,C 180,E1 -4788.761,E2 -4788.761} C_VEL
LIN {X 0,Y 524.79,Z 390.32,A -85,B 0,C 180,E1 -4791.61,E2 -4791.61} C_VEL
LIN {X 0,Y 525.13,Z 375.837,A -85,B 0,C 180,E1 -4794.512,E2 -4794.512} C_VEL
LIN {X 0,Y 523.995,Z 368.839,A -85,B 0,C 180,E1 -4796.021,E2 -4796.021} C_VEL
LIN {X 0,Y 523.947,Z 368.719,A -85,B 0,C 180,E1 -4798.874,E2 -4798.874} C_VEL
LIN {X 0,Y 523.927,Z 368.722,A -85,B 0,C 180,E1 -4801.544,E2 -4801.544} C_VEL
LIN {X 0,Y 523.947,Z 368.721,A -85,B 0,C 180,E1 -4804.289,E2 -4804.289} C_VEL
LIN {X 0,Y 523.914,Z 368.719,A -85,B 0,C 180,E1 -4807.131,E2 -4807.131} C_VEL
LIN {X 0,Y 523.939,Z 368.715,A -85,B 0,C 180,E1 -4810.129,E2 -4810.129} C_VEL
LIN {X 0,Y 523.939,Z 368.719,A -85,B 0,C 180,E1 -4812.459,E2 -4812.459} C_VEL
LIN {X 0,Y 523.957,Z 368.714,A -85,B 0,C 180,E1 -4815.308,E2 -4815.308} C_VEL
LIN {X 0,Y 523.974,Z 368.711,A -85,B 0,C 180,E1 -4818.687,E2 -4818.687} C_VEL
LIN {X 0,Y 523.926,Z 368.716,A -85,B 0,C 180,E1 -4821.079,E2 -4821.079} C_VEL
LIN {X 0,Y 523.925,Z 368.726,A -85,B 0,C 180,E1 -4823.827,E2 -4823.827} C_VEL
LIN {X 0,Y 523.943,Z 368.712,A -85,B 0,C 180,E1 -4826.635,E2 -4826.635} C_VEL
LIN {X 0,Y 523.964,Z 368.715,A -85,B 0,C 180,E1 -4829.356,E2 -4829.356} C_VEL
LIN {X 0,Y 523.979,Z 368.707,A -85,B 0,C 180,E1 -4832.28,E2 -4832.28} C_VEL
LIN {X 0,Y 523.952,Z 368.711,A -85,B 0,C 180,E1 -4834.581,E2 -4834.581} C_VEL
LIN {X 0,Y 523.916,Z 368.719,A -85,B 0,C 180,E1 -4837.106,E2 -4837.106} C_VEL
LIN {X 0,Y 523.978,Z 368.712,A -85,B 0,C 180,E1 -4839.865,E2 -4839.865} C_VEL
LIN {X 0,Y 523.966,Z 368.707,A -85,B 0,C 180,E1 -4842.837,E2 -4842.837} C_VEL
LIN {X 0,Y 523.975,Z 368.712,A -85,B 0,C 180,E1 -4845.235,E2 -4845.235} C_VEL
LIN {X 0,Y 524.011,Z 368.703,A -85,B 0,C 180,E1 -4848.394,E2 -4848.394} C_VEL
LIN {X 0,Y 524.003,Z 368.702,A -85,B 0,C 180,E1 -4851.516,E2 -4851.516} C_VEL
LIN {X 0,Y 524.081,Z 368.698,A -85,B 0,C 180,E1 -4854.613,E2 -4854.613} C_VEL
LIN {X 0,Y 524.109,Z 368.699,A -85,B 0,C 180,E1 -4857.694,E2 -4857.694} C_VEL
LIN {X 0,Y 524.122,Z 368.683,A -85,B 0,C 180,E1 -4860.768,E2 -4860.768} C_VEL
LIN {X 0,Y 524.072,Z 368.698,A -85,B 0,C 180,E1 -4863.074,E2 -4863.074} C_VEL
LIN {X 0,Y 524.043,Z 368.704,A -85,B 0,C 180,E1 -4866.159,E2 -4866.159} C_VEL
LIN {X 0,Y 523.996,Z 368.708,A -85,B 0,C 180,E1 -4869.261,E2 -4869.261} C_VEL
LIN {X 0,Y 524.022,Z 368.71,A -85,B 0,C 180,E1 -4871.751,E2 -4871.751} C_VEL
LIN {X 0,Y 523.989,Z 368.712,A -85,B 0,C 180,E1 -4875.052,E2 -4875.052} C_VEL
LIN {X 0,Y 523.96,Z 368.709,A -85,B 0,C 180,E1 -4877.969,E2 -4877.969} C_VEL
LIN {X 0,Y 523.968,Z 368.708,A -85,B 0,C 180,E1 -4880.41,E2 -4880.41} C_VEL
LIN {X 0,Y 523.913,Z 368.72,A -85,B 0,C 180,E1 -4882.893,E2 -4882.893} C_VEL
LIN {X 0,Y 523.952,Z 368.72,A -85,B 0,C 180,E1 -4885.418,E2 -4885.418} C_VEL
LIN {X 0,Y 523.967,Z 368.71,A -85,B 0,C 180,E1 -4887.998,E2 -4887.998} C_VEL
LIN {X 0,Y 523.943,Z 368.717,A -85,B 0,C 180,E1 -4890.855,E2 -4890.855} C_VEL
LIN {X 0,Y 523.957,Z 368.712,A -85,B 0,C 180,E1 -4893.735,E2 -4893.735} C_VEL
LIN {X 0,Y 523.918,Z 368.718,A -85,B 0,C 180,E1 -4896.404,E2 -4896.404} C_VEL
LIN {X 0,Y 523.919,Z 368.724,A -85,B 0,C 180,E1 -4899.084,E2 -4899.084} C_VEL
LIN {X 0,Y 523.953,Z 368.714,A -85,B 0,C 180,E1 -4902.118,E2 -4902.118} C_VEL
LIN {X 0,Y 523.952,Z 368.718,A -85,B 0,C 180,E1 -4905.308,E2 -4905.308} C_VEL
LIN {X 0,Y 523.915,Z 368.714,A -85,B 0,C 180,E1 -4906.918,E2 -4906.918} C_VEL
LIN {X 0,Y 523.253,Z 368.793,A -85,B 0,C 180,E1 -4907.56,E2 -4907.56} C_VEL
LIN {X 0,Y 520.425,Z 369.145,A -85,B 0,C 180,E1 -4908.602,E2 -4908.602} C_VEL
LIN {X 0,Y 518.027,Z 369.452,A -85,B 0,C 180,E1 -4909.441,E2 -4909.441} C_VEL
LIN {X 0,Y 516.988,Z 369.58,A -85,B 0,C 180,E1 -4910.089,E2 -4910.089} C_VEL
LIN {X 0,Y 516.898,Z 369.591,A -85,B 0,C 180,E1 -4910.308,E2 -4910.308} C_VEL
LIN {X 0,Y 516.881,Z 369.599,A -85,B 0,C 180,E1 -4913.342,E2 -4913.342} C_VEL
LIN {X 0,Y 516.909,Z 369.587,A -85,B 0,C 180,E1 -4916.121,E2 -4916.121} C_VEL
LIN {X 0,Y 516.891,Z 369.6,A -85,B 0,C 180,E1 -4918.935,E2 -4918.935} C_VEL
LIN {X 0,Y 516.921,Z 369.594,A -85,B 0,C 180,E1 -4921.585,E2 -4921.585} C_VEL
LIN {X 0,Y 516.928,Z 369.591,A -85,B 0,C 180,E1 -4924.211,E2 -4924.211} C_VEL
LIN {X 0,Y 516.869,Z 369.602,A -85,B 0,C 180,E1 -4926.776,E2 -4926.776} C_VEL
LIN {X 0,Y 516.936,Z 369.592,A -85,B 0,C 180,E1 -4929.731,E2 -4929.731} C_VEL
LIN {X 0,Y 516.926,Z 369.594,A -85,B 0,C 180,E1 -4932.596,E2 -4932.596} C_VEL
LIN {X 0,Y 516.939,Z 369.596,A -85,B 0,C 180,E1 -4935.03,E2 -4935.03} C_VEL
LIN {X 0,Y 516.962,Z 369.588,A -85,B 0,C 180,E1 -4938.234,E2 -4938.234} C_VEL
LIN {X 0,Y 516.965,Z 369.591,A -85,B 0,C 180,E1 -4941.399,E2 -4941.399} C_VEL
LIN {X 0,Y 517.013,Z 369.582,A -85,B 0,C 180,E1 -4943.757,E2 -4943.757} C_VEL
LIN {X 0,Y 517.082,Z 369.574,A -85,B 0,C 180,E1 -4947.663,E2 -4947.663} C_VEL
LIN {X 0,Y 517.09,Z 369.577,A -85,B 0,C 180,E1 -4950.779,E2 -4950.779} C_VEL
LIN {X 0,Y 517.01,Z 369.587,A -85,B 0,C 180,E1 -4953.117,E2 -4953.117} C_VEL
LIN {X 0,Y 517.013,Z 369.582,A -85,B 0,C 180,E1 -4956.243,E2 -4956.243} C_VEL
LIN {X 0,Y 516.951,Z 369.592,A -85,B 0,C 180,E1 -4959.389,E2 -4959.389} C_VEL
LIN {X 0,Y 516.948,Z 369.589,A -85,B 0,C 180,E1 -4961.807,E2 -4961.807} C_VEL
LIN {X 0,Y 516.94,Z 369.595,A -85,B 0,C 180,E1 -4965.146,E2 -4965.146} C_VEL
LIN {X 0,Y 516.922,Z 369.593,A -85,B 0,C 180,E1 -4968.222,E2 -4968.222} C_VEL
LIN {X 0,Y 516.908,Z 369.6,A -85,B 0,C 180,E1 -4970.701,E2 -4970.701} C_VEL
LIN {X 0,Y 516.906,Z 369.594,A -85,B 0,C 180,E1 -4974.072,E2 -4974.072} C_VEL
LIN {X 0,Y 516.924,Z 369.598,A -85,B 0,C 180,E1 -4976.657,E2 -4976.657} C_VEL
LIN {X 0,Y 516.92,Z 369.587,A -85,B 0,C 180,E1 -4979.526,E2 -4979.526} C_VEL
LIN {X 0,Y 516.895,Z 369.6,A -85,B 0,C 180,E1 -4982.544,E2 -4982.544} C_VEL
LIN {X 0,Y 516.877,Z 369.593,A -85,B 0,C 180,E1 -4985.332,E2 -4985.332} C_VEL
LIN {X 0,Y 516.876,Z 369.597,A -85,B 0,C 180,E1 -4987.943,E2 -4987.943} C_VEL
LIN {X 0,Y 516.897,Z 369.588,A -85,B 0,C 180,E1 -4990.739,E2 -4990.739} C_VEL
LIN {X 0,Y 516.875,Z 369.59,A -85,B 0,C 180,E1 -4993.903,E2 -4993.903} C_VEL
LIN {X 0,Y 516.876,Z 369.597,A -85,B 0,C 180,E1 -4996.107,E2 -4996.107} C_VEL
LIN {X 0,Y 516.91,Z 369.596,A -85,B 0,C 180,E1 -4998.398,E2 -4998.398} C_VEL
LIN {X 0,Y 516.876,Z 369.597,A -85,B 0,C 180,E1 -5001.284,E2 -5001.284} C_VEL
LIN {X 0,Y 516.884,Z 369.598,A -85,B 0,C 180,E1 -5004.221,E2 -5004.221} C_VEL
LIN {X 0,Y 516.891,Z 369.596,A -85,B 0,C 180,E1 -5007.053,E2 -5007.053} C_VEL
LIN {X 0,Y 516.895,Z 369.594,A -85,B 0,C 180,E1 -5009.797,E2 -5009.797} C_VEL
LIN {X 0,Y 516.923,Z 369.59,A -85,B 0,C 180,E1 -5012.468,E2 -5012.468} C_VEL
LIN {X 0,Y 516.905,Z 369.594,A -85,B 0,C 180,E1 -5015.072,E2 -5015.072} C_VEL
LIN {X 0,Y 516.88,Z 369.601,A -85,B 0,C 180,E1 -5018.463,E2 -5018.463} C_VEL
LIN {X 0,Y 516.898,Z 369.588,A -85,B 0,C 180,E1 -5020.955,E2 -5020.955} C_VEL
LIN {X 0,Y 516.911,Z 369.59,A -85,B 0,C 180,E1 -5023.411,E2 -5023.411} C_VEL
LIN {X 0,Y 516.889,Z 369.596,A -85,B 0,C 180,E1 -5025.834,E2 -5025.834} C_VEL
LIN {X 0,Y 516.997,Z 369.584,A -85,B 0,C 180,E1 -5028.235,E2 -5028.235} C_VEL
LIN {X 0,Y 516.963,Z 369.579,A -85,B 0,C 180,E1 -5031.4,E2 -5031.4} C_VEL
LIN {X 0,Y 517.004,Z 369.58,A -85,B 0,C 180,E1 -5033.757,E2 -5033.757} C_VEL
LIN {X 0,Y 517.079,Z 369.568,A -85,B 0,C 180,E1 -5037.664,E2 -5037.664} C_VEL
LIN {X 0,Y 517.089,Z 369.567,A -85,B 0,C 180,E1 -5040.779,E2 -5040.779} C_VEL
LIN {X 0,Y 517.01,Z 369.579,A -85,B 0,C 180,E1 -5043.117,E2 -5043.117} C_VEL
LIN {X 0,Y 517.005,Z 369.587,A -85,B 0,C 180,E1 -5046.244,E2 -5046.244} C_VEL
LIN {X 0,Y 516.949,Z 369.575,A -85,B 0,C 180,E1 -5049.39,E2 -5049.39} C_VEL
LIN {X 0,Y 516.946,Z 369.585,A -85,B 0,C 180,E1 -5051.808,E2 -5051.808} C_VEL
LIN {X 0,Y 516.939,Z 369.586,A -85,B 0,C 180,E1 -5055.147,E2 -5055.147} C_VEL
LIN {X 0,Y 516.921,Z 369.588,A -85,B 0,C 180,E1 -5058.223,E2 -5058.223} C_VEL
LIN {X 0,Y 516.909,Z 369.592,A -85,B 0,C 180,E1 -5060.702,E2 -5060.702} C_VEL
LIN {X 0,Y 516.907,Z 369.599,A -85,B 0,C 180,E1 -5064.073,E2 -5064.073} C_VEL
LIN {X 0,Y 516.925,Z 369.585,A -85,B 0,C 180,E1 -5066.658,E2 -5066.658} C_VEL
LIN {X 0,Y 516.921,Z 369.59,A -85,B 0,C 180,E1 -5069.527,E2 -5069.527} C_VEL
LIN {X 0,Y 516.898,Z 369.592,A -85,B 0,C 180,E1 -5072.545,E2 -5072.545} C_VEL
LIN {X 0,Y 516.88,Z 369.593,A -85,B 0,C 180,E1 -5075.333,E2 -5075.333} C_VEL
LIN {X 0,Y 516.879,Z 369.603,A -85,B 0,C 180,E1 -5077.944,E2 -5077.944} C_VEL
LIN {X 0,Y 516.902,Z 369.593,A -85,B 0,C 180,E1 -5080.74,E2 -5080.74} C_VEL
LIN {X 0,Y 516.881,Z 369.602,A -85,B 0,C 180,E1 -5083.904,E2 -5083.904} C_VEL
LIN {X 0,Y 516.881,Z 369.603,A -85,B 0,C 180,E1 -5086.108,E2 -5086.108} C_VEL
LIN {X 0,Y 516.916,Z 369.587,A -85,B 0,C 180,E1 -5088.399,E2 -5088.399} C_VEL
LIN {X 0,Y 516.883,Z 369.596,A -85,B 0,C 180,E1 -5091.285,E2 -5091.285} C_VEL
LIN {X 0,Y 516.891,Z 369.597,A -85,B 0,C 180,E1 -5094.222,E2 -5094.222} C_VEL
LIN {X 0,Y 516.897,Z 369.592,A -85,B 0,C 180,E1 -5097.054,E2 -5097.054} C_VEL
LIN {X 0,Y 516.903,Z 369.598,A -85,B 0,C 180,E1 -5099.798,E2 -5099.798} C_VEL
LIN {X 0,Y 516.93,Z 369.596,A -85,B 0,C 180,E1 -5102.468,E2 -5102.468} C_VEL
LIN {X 0,Y 517.002,Z 369.831,A -85,B 0,C 180,E1 -5103.841,E2 -5103.841} C_VEL
LIN {X 0,Y 518.126,Z 376.699,A -85,B 0,C 180,E1 -5105.341,E2 -5105.341} C_VEL
LIN {X 0,Y 517.906,Z 388.114,A -85,B 0,C 180,E1 -5107.669,E2 -5107.669} C_VEL
LIN {X 0,Y 517.545,Z 401.697,A -85,B 0,C 180,E1 -5110.362,E2 -5110.362} C_VEL
LIN {X 0,Y 517.258,Z 414.197,A -85,B 0,C 180,E1 -5112.812,E2 -5112.812} C_VEL
LIN {X 0,Y 517.053,Z 423.44,A -85,B 0,C 180,E1 -5114.608,E2 -5114.608} C_VEL
LIN {X 0,Y 517.811,Z 428.378,A -85,B 0,C 180,E1 -5114.739,E2 -5114.739} C_VEL
LIN {X 0,Y 519.094,Z 436.524,A -85,B 0,C 180,E1 -5114.891,E2 -5114.891} C_VEL
LIN {X 0,Y 518.657,Z 528.417,A -85,B 0,C 180,E1 -5116.183,E2 -5116.183} C_VEL
LIN {X 0,Y 518.482,Z 538.331,A -85,B 0,C 180,E1 -5116.403,E2 -5116.403} C_VEL
LIN {X 0,Y 518.32,Z 548.32,A -85,B 0,C 180,E1 -5116.723,E2 -5116.723} C_VEL
LIN {X 0,Y 518.038,Z 558.678,A -85,B 0,C 180,E1 -5117.165,E2 -5117.165} C_VEL
LIN {X 0,Y 517.83,Z 568.294,A -85,B 0,C 180,E1 -5117.687,E2 -5117.687} C_VEL
LIN {X 0,Y 517.597,Z 576.834,A -85,B 0,C 180,E1 -5118.249,E2 -5118.249} C_VEL
LIN {X 0,Y 517.346,Z 585.565,A -85,B 0,C 180,E1 -5118.938,E2 -5118.938} C_VEL
LIN {X 0,Y 517.134,Z 592.989,A -85,B 0,C 180,E1 -5119.626,E2 -5119.626} C_VEL
LIN {X 0,Y 516.856,Z 601.787,A -85,B 0,C 180,E1 -5120.609,E2 -5120.609} C_VEL
LIN {X 0,Y 516.728,Z 607.779,A -85,B 0,C 180,E1 -5121.396,E2 -5121.396} C_VEL
LIN {X 0,Y 516.557,Z 614.089,A -85,B 0,C 180,E1 -5122.377,E2 -5122.377} C_VEL
LIN {X 0,Y 516.452,Z 619.63,A -85,B 0,C 180,E1 -5123.417,E2 -5123.417} C_VEL
LIN {X 0,Y 516.378,Z 624.452,A -85,B 0,C 180,E1 -5124.533,E2 -5124.533} C_VEL
LIN {X 0,Y 516.313,Z 628.41,A -85,B 0,C 180,E1 -5125.707,E2 -5125.707} C_VEL
LIN {X 0,Y 516.282,Z 631.338,A -85,B 0,C 180,E1 -5126.879,E2 -5126.879} C_VEL
LIN {X 0,Y 516.261,Z 632.834,A -85,B 0,C 180,E1 -5127.66,E2 -5127.66} C_VEL
LIN {X 0,Y 516.16,Z 634.349,A -85,B 0,C 180,E1 -5129.22,E2 -5129.22} C_VEL
LIN {X 0,Y 516.154,Z 634.627,A -85,B 0,C 180,E1 -5130,E2 -5130} C_VEL
LIN {X 0,Y 516.192,Z 633.756,A -85,B 0,C 180,E1 -5131.561,E2 -5131.561} C_VEL
LIN {X 0,Y 516.261,Z 632.833,A -85,B 0,C 180,E1 -5132.341,E2 -5132.341} C_VEL
LIN {X 0,Y 516.352,Z 629.497,A -85,B 0,C 180,E1 -5133.902,E2 -5133.902} C_VEL
LIN {X 0,Y 516.313,Z 625.875,A -85,B 0,C 180,E1 -5135.076,E2 -5135.076} C_VEL
LIN {X 0,Y 516.427,Z 622.938,A -85,B 0,C 180,E1 -5135.858,E2 -5135.858} C_VEL
LIN {X 0,Y 516.51,Z 617.364,A -85,B 0,C 180,E1 -5137.034,E2 -5137.034} C_VEL
LIN {X 0,Y 516.631,Z 611.712,A -85,B 0,C 180,E1 -5138.015,E2 -5138.015} C_VEL
LIN {X 0,Y 516.783,Z 604.906,A -85,B 0,C 180,E1 -5138.998,E2 -5138.998} C_VEL
LIN {X 0,Y 517.026,Z 596.687,A -85,B 0,C 180,E1 -5139.981,E2 -5139.981} C_VEL
LIN {X 0,Y 517.27,Z 588.857,A -85,B 0,C 180,E1 -5140.767,E2 -5140.767} C_VEL
LIN {X 0,Y 517.524,Z 580.77,A -85,B 0,C 180,E1 -5141.456,E2 -5141.456} C_VEL
LIN {X 0,Y 517.756,Z 570.958,A -85,B 0,C 180,E1 -5142.148,E2 -5142.148} C_VEL
LIN {X 0,Y 517.978,Z 562.608,A -85,B 0,C 180,E1 -5142.638,E2 -5142.638} C_VEL
LIN {X 0,Y 518.225,Z 552.097,A -85,B 0,C 180,E1 -5143.13,E2 -5143.13} C_VEL
LIN {X 0,Y 518.419,Z 541.759,A -85,B 0,C 180,E1 -5143.499,E2 -5143.499} C_VEL
LIN {X 0,Y 518.626,Z 531.035,A -85,B 0,C 180,E1 -5143.768,E2 -5143.768} C_VEL
LIN {X 0,Y 518.821,Z 508.257,A -85,B 0,C 180,E1 -5144.113,E2 -5144.113} C_VEL
LIN {X 0,Y 518.955,Z 434.793,A -85,B 0,C 180,E1 -5145.137,E2 -5145.137} C_VEL
LIN {X 0,Y 517.115,Z 423.87,A -85,B 0,C 180,E1 -5145.36,E2 -5145.36} C_VEL
LIN {X 0,Y 517.079,Z 422.515,A -85,B 0,C 180,E1 -5145.548,E2 -5145.548} C_VEL
LIN {X 0,Y 517.477,Z 406.923,A -85,B 0,C 180,E1 -5148.612,E2 -5148.612} C_VEL
LIN {X 0,Y 517.823,Z 391.231,A -85,B 0,C 180,E1 -5151.706,E2 -5151.706} C_VEL
LIN {X 0,Y 518.204,Z 378.245,A -85,B 0,C 180,E1 -5154.336,E2 -5154.336} C_VEL
LIN {X 0,Y 517.669,Z 373.637,A -85,B 0,C 180,E1 -5155.319,E2 -5155.319} C_VEL
LIN {X 0,Y 516.976,Z 369.717,A -85,B 0,C 180,E1 -5156.203,E2 -5156.203} C_VEL
LIN {X 0,Y 516.933,Z 369.593,A -85,B 0,C 180,E1 -5159.304,E2 -5159.304} C_VEL
LIN {X 0,Y 516.9,Z 369.595,A -85,B 0,C 180,E1 -5162.543,E2 -5162.543} C_VEL
LIN {X 0,Y 516.886,Z 369.596,A -85,B 0,C 180,E1 -5165.332,E2 -5165.332} C_VEL
LIN {X 0,Y 516.884,Z 369.602,A -85,B 0,C 180,E1 -5167.943,E2 -5167.943} C_VEL
LIN {X 0,Y 516.887,Z 369.588,A -85,B 0,C 180,E1 -5170.741,E2 -5170.741} C_VEL
LIN {X 0,Y 516.886,Z 369.595,A -85,B 0,C 180,E1 -5172.831,E2 -5172.831} C_VEL
LIN {X 0,Y 516.924,Z 369.589,A -85,B 0,C 180,E1 -5175.01,E2 -5175.01} C_VEL
LIN {X 0,Y 516.924,Z 369.592,A -85,B 0,C 180,E1 -5178.397,E2 -5178.397} C_VEL
LIN {X 0,Y 516.887,Z 369.593,A -85,B 0,C 180,E1 -5181.284,E2 -5181.284} C_VEL
LIN {X 0,Y 516.888,Z 369.596,A -85,B 0,C 180,E1 -5184.221,E2 -5184.221} C_VEL
LIN {X 0,Y 516.898,Z 369.589,A -85,B 0,C 180,E1 -5187.053,E2 -5187.053} C_VEL
LIN {X 0,Y 516.902,Z 369.601,A -85,B 0,C 180,E1 -5189.797,E2 -5189.797} C_VEL
LIN {X 0,Y 516.928,Z 369.584,A -85,B 0,C 180,E1 -5192.467,E2 -5192.467} C_VEL
LIN {X 0,Y 516.91,Z 369.588,A -85,B 0,C 180,E1 -5195.071,E2 -5195.071} C_VEL
LIN {X 0,Y 516.869,Z 369.602,A -85,B 0,C 180,E1 -5197.621,E2 -5197.621} C_VEL
LIN {X 0,Y 516.931,Z 369.585,A -85,B 0,C 180,E1 -5200.129,E2 -5200.129} C_VEL
LIN {X 0,Y 516.928,Z 369.583,A -85,B 0,C 180,E1 -5202.596,E2 -5202.596} C_VEL
LIN {X 0,Y 516.94,Z 369.587,A -85,B 0,C 180,E1 -5205.03,E2 -5205.03} C_VEL
LIN {X 0,Y 516.964,Z 369.582,A -85,B 0,C 180,E1 -5208.233,E2 -5208.233} C_VEL
LIN {X 0,Y 516.968,Z 369.576,A -85,B 0,C 180,E1 -5211.399,E2 -5211.399} C_VEL
LIN {X 0,Y 517.008,Z 369.586,A -85,B 0,C 180,E1 -5213.756,E2 -5213.756} C_VEL
LIN {X 0,Y 517.081,Z 369.575,A -85,B 0,C 180,E1 -5217.663,E2 -5217.663} C_VEL
LIN {X 0,Y 517.092,Z 369.558,A -85,B 0,C 180,E1 -5220.778,E2 -5220.778} C_VEL
LIN {X 0,Y 517.013,Z 369.577,A -85,B 0,C 180,E1 -5223.116,E2 -5223.116} C_VEL
LIN {X 0,Y 517.007,Z 369.58,A -85,B 0,C 180,E1 -5226.243,E2 -5226.243} C_VEL
LIN {X 0,Y 516.95,Z 369.586,A -85,B 0,C 180,E1 -5229.389,E2 -5229.389} C_VEL
LIN {X 0,Y 516.98,Z 369.585,A -85,B 0,C 180,E1 -5231.824,E2 -5231.824} C_VEL
LIN {X 0,Y 516.941,Z 369.591,A -85,B 0,C 180,E1 -5235.146,E2 -5235.146} C_VEL
LIN {X 0,Y 516.922,Z 369.583,A -85,B 0,C 180,E1 -5238.222,E2 -5238.222} C_VEL
LIN {X 0,Y 516.909,Z 369.587,A -85,B 0,C 180,E1 -5240.701,E2 -5240.701} C_VEL
LIN {X 0,Y 516.908,Z 369.593,A -85,B 0,C 180,E1 -5244.072,E2 -5244.072} C_VEL
LIN {X 0,Y 516.925,Z 369.585,A -85,B 0,C 180,E1 -5246.657,E2 -5246.657} C_VEL
LIN {X 0,Y 516.907,Z 369.599,A -85,B 0,C 180,E1 -5249.524,E2 -5249.524} C_VEL
LIN {X 0,Y 516.897,Z 369.593,A -85,B 0,C 180,E1 -5252.544,E2 -5252.544} C_VEL
LIN {X 0,Y 516.879,Z 369.597,A -85,B 0,C 180,E1 -5255.332,E2 -5255.332} C_VEL
LIN {X 0,Y 516.877,Z 369.598,A -85,B 0,C 180,E1 -5257.943,E2 -5257.943} C_VEL
LIN {X 0,Y 516.882,Z 369.592,A -85,B 0,C 180,E1 -5260.741,E2 -5260.741} C_VEL
LIN {X 0,Y 516.901,Z 369.594,A -85,B 0,C 180,E1 -5262.829,E2 -5262.829} C_VEL
LIN {X 0,Y 516.918,Z 369.595,A -85,B 0,C 180,E1 -5265.01,E2 -5265.01} C_VEL
LIN {X 0,Y 516.918,Z 369.577,A -85,B 0,C 180,E1 -5268.397,E2 -5268.397} C_VEL
LIN {X 0,Y 516.898,Z 369.591,A -85,B 0,C 180,E1 -5270.308,E2 -5270.308} C_VEL
LIN {X 0,Y 516.217,Z 369.681,A -85,B 0,C 180,E1 -5270.958,E2 -5270.958} C_VEL
LIN {X 0,Y 513.363,Z 370.037,A -85,B 0,C 180,E1 -5272.014,E2 -5272.014} C_VEL
LIN {X 0,Y 510.955,Z 370.338,A -85,B 0,C 180,E1 -5272.864,E2 -5272.864} C_VEL
LIN {X 0,Y 509.916,Z 370.464,A -85,B 0,C 180,E1 -5273.52,E2 -5273.52} C_VEL
LIN {X 0,Y 509.828,Z 370.472,A -85,B 0,C 180,E1 -5273.742,E2 -5273.742} C_VEL
LIN {X 0,Y 509.859,Z 370.466,A -85,B 0,C 180,E1 -5276.539,E2 -5276.539} C_VEL
LIN {X 0,Y 509.848,Z 370.474,A -85,B 0,C 180,E1 -5279.335,E2 -5279.335} C_VEL
LIN {X 0,Y 509.891,Z 370.467,A -85,B 0,C 180,E1 -5282.055,E2 -5282.055} C_VEL
LIN {X 0,Y 509.874,Z 370.472,A -85,B 0,C 180,E1 -5284.704,E2 -5284.704} C_VEL
LIN {X 0,Y 509.853,Z 370.477,A -85,B 0,C 180,E1 -5287.45,E2 -5287.45} C_VEL
LIN {X 0,Y 509.913,Z 370.466,A -85,B 0,C 180,E1 -5289.845,E2 -5289.845} C_VEL
LIN {X 0,Y 509.881,Z 370.476,A -85,B 0,C 180,E1 -5293.175,E2 -5293.175} C_VEL
LIN {X 0,Y 509.861,Z 370.474,A -85,B 0,C 180,E1 -5295.634,E2 -5295.634} C_VEL
LIN {X 0,Y 509.91,Z 370.471,A -85,B 0,C 180,E1 -5298.874,E2 -5298.874} C_VEL
LIN {X 0,Y 509.948,Z 370.462,A -85,B 0,C 180,E1 -5302.078,E2 -5302.078} C_VEL
LIN {X 0,Y 509.983,Z 370.459,A -85,B 0,C 180,E1 -5304.464,E2 -5304.464} C_VEL
LIN {X 0,Y 510.053,Z 370.45,A -85,B 0,C 180,E1 -5307.631,E2 -5307.631} C_VEL
LIN {X 0,Y 510.061,Z 370.452,A -85,B 0,C 180,E1 -5310.789,E2 -5310.789} C_VEL
LIN {X 0,Y 509.952,Z 370.466,A -85,B 0,C 180,E1 -5313.16,E2 -5313.16} C_VEL
LIN {X 0,Y 509.98,Z 370.459,A -85,B 0,C 180,E1 -5316.329,E2 -5316.329} C_VEL
LIN {X 0,Y 509.913,Z 370.471,A -85,B 0,C 180,E1 -5318.72,E2 -5318.72} C_VEL
LIN {X 0,Y 509.9,Z 370.467,A -85,B 0,C 180,E1 -5321.931,E2 -5321.931} C_VEL
LIN {X 0,Y 509.889,Z 370.472,A -85,B 0,C 180,E1 -5325.241,E2 -5325.241} C_VEL
LIN {X 0,Y 509.884,Z 370.469,A -85,B 0,C 180,E1 -5328.001,E2 -5328.001} C_VEL
LIN {X 0,Y 509.846,Z 370.48,A -85,B 0,C 180,E1 -5331.001,E2 -5331.001} C_VEL
LIN {X 0,Y 509.832,Z 370.476,A -85,B 0,C 180,E1 -5333.563,E2 -5333.563} C_VEL
LIN {X 0,Y 509.909,Z 370.468,A -85,B 0,C 180,E1 -5336.379,E2 -5336.379} C_VEL
LIN {X 0,Y 509.881,Z 370.468,A -85,B 0,C 180,E1 -5338.843,E2 -5338.843} C_VEL
LIN {X 0,Y 509.821,Z 370.476,A -85,B 0,C 180,E1 -5341.589,E2 -5341.589} C_VEL
LIN {X 0,Y 509.848,Z 370.469,A -85,B 0,C 180,E1 -5344.413,E2 -5344.413} C_VEL
LIN {X 0,Y 509.813,Z 370.478,A -85,B 0,C 180,E1 -5347.34,E2 -5347.34} C_VEL
LIN {X 0,Y 509.854,Z 370.472,A -85,B 0,C 180,E1 -5350.38,E2 -5350.38} C_VEL
LIN {X 0,Y 509.817,Z 370.472,A -85,B 0,C 180,E1 -5353.062,E2 -5353.062} C_VEL
LIN {X 0,Y 509.824,Z 370.474,A -85,B 0,C 180,E1 -5355.792,E2 -5355.792} C_VEL
LIN {X 0,Y 509.852,Z 370.475,A -85,B 0,C 180,E1 -5358.575,E2 -5358.575} C_VEL
LIN {X 0,Y 509.846,Z 370.472,A -85,B 0,C 180,E1 -5361.786,E2 -5361.786} C_VEL
LIN {X 0,Y 509.839,Z 370.474,A -85,B 0,C 180,E1 -5364.623,E2 -5364.623} C_VEL
LIN {X 0,Y 509.859,Z 370.469,A -85,B 0,C 180,E1 -5367.481,E2 -5367.481} C_VEL
LIN {X 0,Y 509.874,Z 370.473,A -85,B 0,C 180,E1 -5370.269,E2 -5370.269} C_VEL
LIN {X 0,Y 509.88,Z 370.465,A -85,B 0,C 180,E1 -5372.945,E2 -5372.945} C_VEL
LIN {X 0,Y 509.863,Z 370.469,A -85,B 0,C 180,E1 -5375.574,E2 -5375.574} C_VEL
LIN {X 0,Y 509.816,Z 370.479,A -85,B 0,C 180,E1 -5378.149,E2 -5378.149} C_VEL
LIN {X 0,Y 509.858,Z 370.467,A -85,B 0,C 180,E1 -5380.682,E2 -5380.682} C_VEL
LIN {X 0,Y 509.88,Z 370.466,A -85,B 0,C 180,E1 -5383.175,E2 -5383.175} C_VEL
LIN {X 0,Y 509.857,Z 370.47,A -85,B 0,C 180,E1 -5385.634,E2 -5385.634} C_VEL
LIN {X 0,Y 509.916,Z 370.456,A -85,B 0,C 180,E1 -5388.875,E2 -5388.875} C_VEL
LIN {X 0,Y 509.945,Z 370.457,A -85,B 0,C 180,E1 -5392.079,E2 -5392.079} C_VEL
LIN {X 0,Y 509.977,Z 370.463,A -85,B 0,C 180,E1 -5394.465,E2 -5394.465} C_VEL
LIN {X 0,Y 510.05,Z 370.443,A -85,B 0,C 180,E1 -5397.631,E2 -5397.631} C_VEL
LIN {X 0,Y 510.059,Z 370.442,A -85,B 0,C 180,E1 -5400.79,E2 -5400.79} C_VEL
LIN {X 0,Y 509.952,Z 370.458,A -85,B 0,C 180,E1 -5403.161,E2 -5403.161} C_VEL
LIN {X 0,Y 509.973,Z 370.46,A -85,B 0,C 180,E1 -5406.33,E2 -5406.33} C_VEL
LIN {X 0,Y 509.911,Z 370.454,A -85,B 0,C 180,E1 -5408.721,E2 -5408.721} C_VEL
LIN {X 0,Y 509.898,Z 370.464,A -85,B 0,C 180,E1 -5411.932,E2 -5411.932} C_VEL
LIN {X 0,Y 509.888,Z 370.465,A -85,B 0,C 180,E1 -5415.242,E2 -5415.242} C_VEL
LIN {X 0,Y 509.884,Z 370.465,A -85,B 0,C 180,E1 -5418.002,E2 -5418.002} C_VEL
LIN {X 0,Y 509.846,Z 370.47,A -85,B 0,C 180,E1 -5421.002,E2 -5421.002} C_VEL
LIN {X 0,Y 509.832,Z 370.474,A -85,B 0,C 180,E1 -5423.564,E2 -5423.564} C_VEL
LIN {X 0,Y 509.91,Z 370.461,A -85,B 0,C 180,E1 -5426.38,E2 -5426.38} C_VEL
LIN {X 0,Y 509.882,Z 370.467,A -85,B 0,C 180,E1 -5428.844,E2 -5428.844} C_VEL
LIN {X 0,Y 509.824,Z 370.476,A -85,B 0,C 180,E1 -5431.59,E2 -5431.59} C_VEL
LIN {X 0,Y 509.852,Z 370.472,A -85,B 0,C 180,E1 -5434.414,E2 -5434.414} C_VEL
LIN {X 0,Y 509.817,Z 370.476,A -85,B 0,C 180,E1 -5437.341,E2 -5437.341} C_VEL
LIN {X 0,Y 509.859,Z 370.473,A -85,B 0,C 180,E1 -5440.381,E2 -5440.381} C_VEL
LIN {X 0,Y 509.838,Z 370.472,A -85,B 0,C 180,E1 -5443.065,E2 -5443.065} C_VEL
LIN {X 0,Y 509.829,Z 370.479,A -85,B 0,C 180,E1 -5445.793,E2 -5445.793} C_VEL
LIN {X 0,Y 509.857,Z 370.464,A -85,B 0,C 180,E1 -5448.576,E2 -5448.576} C_VEL
LIN {X 0,Y 509.851,Z 370.477,A -85,B 0,C 180,E1 -5451.787,E2 -5451.787} C_VEL
LIN {X 0,Y 509.847,Z 370.472,A -85,B 0,C 180,E1 -5454.624,E2 -5454.624} C_VEL
LIN {X 0,Y 509.864,Z 370.471,A -85,B 0,C 180,E1 -5457.482,E2 -5457.482} C_VEL
LIN {X 0,Y 509.883,Z 370.473,A -85,B 0,C 180,E1 -5460.27,E2 -5460.27} C_VEL
LIN {X 0,Y 509.89,Z 370.472,A -85,B 0,C 180,E1 -5462.945,E2 -5462.945} C_VEL
LIN {X 0,Y 509.966,Z 370.7,A -85,B 0,C 180,E1 -5463.66,E2 -5463.66} C_VEL
LIN {X 0,Y 511.212,Z 378.571,A -85,B 0,C 180,E1 -5465.406,E2 -5465.406} C_VEL
LIN {X 0,Y 510.865,Z 392.144,A -85,B 0,C 180,E1 -5468.196,E2 -5468.196} C_VEL
LIN {X 0,Y 510.45,Z 408.868,A -85,B 0,C 180,E1 -5471.539,E2 -5471.539} C_VEL
LIN {X 0,Y 510.026,Z 423.228,A -85,B 0,C 180,E1 -5474.39,E2 -5474.39} C_VEL
LIN {X 0,Y 510.765,Z 427.918,A -85,B 0,C 180,E1 -5474.519,E2 -5474.519} C_VEL
LIN {X 0,Y 512.24,Z 437.474,A -85,B 0,C 180,E1 -5474.7,E2 -5474.7} C_VEL
LIN {X 0,Y 511.771,Z 528.222,A -85,B 0,C 180,E1 -5475.994,E2 -5475.994} C_VEL
LIN {X 0,Y 511.584,Z 538.136,A -85,B 0,C 180,E1 -5476.216,E2 -5476.216} C_VEL
LIN {X 0,Y 511.411,Z 548.125,A -85,B 0,C 180,E1 -5476.541,E2 -5476.541} C_VEL
LIN {X 0,Y 511.103,Z 558.483,A -85,B 0,C 180,E1 -5476.988,E2 -5476.988} C_VEL
LIN {X 0,Y 510.862,Z 567.958,A -85,B 0,C 180,E1 -5477.507,E2 -5477.507} C_VEL
LIN {X 0,Y 510.64,Z 576.639,A -85,B 0,C 180,E1 -5478.086,E2 -5478.086} C_VEL
LIN {X 0,Y 510.337,Z 585.369,A -85,B 0,C 180,E1 -5478.784,E2 -5478.784} C_VEL
LIN {X 0,Y 510.095,Z 592.793,A -85,B 0,C 180,E1 -5479.482,E2 -5479.482} C_VEL
LIN {X 0,Y 509.829,Z 601.592,A -85,B 0,C 180,E1 -5480.479,E2 -5480.479} C_VEL
LIN {X 0,Y 509.665,Z 607.583,A -85,B 0,C 180,E1 -5481.276,E2 -5481.276} C_VEL
LIN {X 0,Y 509.488,Z 613.894,A -85,B 0,C 180,E1 -5482.271,E2 -5482.271} C_VEL
LIN {X 0,Y 509.35,Z 619.968,A -85,B 0,C 180,E1 -5483.443,E2 -5483.443} C_VEL
LIN {X 0,Y 509.296,Z 624.256,A -85,B 0,C 180,E1 -5484.457,E2 -5484.457} C_VEL
LIN {X 0,Y 509.205,Z 628.214,A -85,B 0,C 180,E1 -5485.647,E2 -5485.647} C_VEL
LIN {X 0,Y 509.2,Z 631.143,A -85,B 0,C 180,E1 -5486.835,E2 -5486.835} C_VEL
LIN {X 0,Y 509.189,Z 632.64,A -85,B 0,C 180,E1 -5487.627,E2 -5487.627} C_VEL
LIN {X 0,Y 509.073,Z 634.154,A -85,B 0,C 180,E1 -5489.209,E2 -5489.209} C_VEL
LIN {X 0,Y 509.065,Z 634.432,A -85,B 0,C 180,E1 -5490,E2 -5490} C_VEL
LIN {X 0,Y 509.112,Z 633.562,A -85,B 0,C 180,E1 -5491.582,E2 -5491.582} C_VEL
LIN {X 0,Y 509.19,Z 632.639,A -85,B 0,C 180,E1 -5492.373,E2 -5492.373} C_VEL
LIN {X 0,Y 509.246,Z 629.301,A -85,B 0,C 180,E1 -5493.957,E2 -5493.957} C_VEL
LIN {X 0,Y 509.244,Z 625.68,A -85,B 0,C 180,E1 -5495.147,E2 -5495.147} C_VEL
